(* CODESYS project Rasi_feeds_batching.project

Project tree, tasks and I/O mapping:
  PLC_AC500_V3 : PM5032-T-ETH, ABB AG, order no. 1SAP123400R0x72, version 3.7.0.0
    application Application
      task Task (cyclic, interval t#10ms, priority 14, watchdog t#20ms x 1) calls batching14
      CheckConfigurationObject
      old_version/
        program batching1 [ST]
        program batching2 [ST]
        program batching3 [ST]
        program batching4 [ST]
        program batching5 [ST]
        function block Auto_Batching [ST]
        function block Manual_Batching [ST]
        program batching6 [ST]
        function block Auto_Batching_V7 [ST]
        function block Manual_Batching_V7 [ST]
        program batching7 [ST]
        function block Auto_Batching_V8 [ST]
        function block Manual_Batching_V8 [ST]
        program batching8 [ST]
        function block Auto_Batching_V9 [ST]
        function block Manual_Batching_V9 [ST]
        program batching9 [ST]
        function block Auto_Batching_V10 [ST]
        function block Manual_Batching_V10 [ST]
        program batching10 [ST]
        program batching11 [ST]
        function block Auto_Batching_V11 [ST]
        function block Semi_Auto_Batching_V11 [ST]
        function block Auto_Batching_V12 [ST]
        function block Semi_Auto_Batching_V12 [ST]
        program batching12 [ST]
      Diagnosis/
        text list Diag_IO_Bus
        text list Diag_V3_PLC
      global variables GVL
      function block Auto_Batching_V13 [ST]
      function block Semi_Auto_Batching_V13 [ST]
      program batching13 [ST]
      function block Auto_Batching_V14 [ST]
      function block Semi_Auto_Batching_V14 [ST]
      program batching14 [FBD]
    OnBoard_IO : 12DI/8DO-T/2DC, ABB AG, version 3.7.0.0
        unmapped channels: Fast inputs DI0-DI3, Fast inputs DI4-DI7, Standard inputs DI8-DI11, Digital inputs - Transistor, Fast outputs DO0-DO3, Fast outputs DO4-DO7, Digital outputs - Transistor
    IO_Bus : I/O-Bus, ABB AG, version 3.7.0.0
    Interfaces : Interfaces, ABB AG, version 3.7.0.0
      OptionSlot_1
      OptionSlot_2
      Ethernet : Ethernet, ABB AG, version 3.7.0.0
        ETH1 : IP Settings, ABB AG, version 3.7.0.0
          NetConfig : NetConfig, ABB AG, version 3.7.0.0
          Modbus_TCP_IP_Server : Modbus TCP/IP Server, ABB AG, version 3.7.0.0
        Protocols : Client Protocols, ABB AG, version 3.7.0.0
    OnBoard_RTC : OnBoard RTC, ABB AG, version 3.7.0.0
  text list GlobalTextList
*)

// PLC_AC500_V3/Application/GVL
{attribute 'qualified_only'}
VAR_GLOBAL
    Recipe_Weights AT %MD100 : ARRAY[1..20] OF REAL;
	Auto_Bin_Material_Mapping AT %MW50: ARRAY[1..6] OF INT;
	Semi_Auto_Bin_Material_Mapping AT %MW60: ARRAY[1..10] OF INT;
	Auto_Bin_Cutoff_Weights AT %MD120: ARRAY[1..6] OF REAL;
	Semi_Auto_Bin_Cutoff_Weights AT %MD130: ARRAY[1..10] OF REAL;
	Auto_Bin_Tolerance AT %MD150: ARRAY[1..6] OF REAL;
	Semi_Auto_Bin_Tolerance AT %MD160: ARRAY[1..10] OF REAL;
	Start_Button AT %MX2.0: BOOL;
	E_Stop_Active AT %MX2.1: BOOL;
	Reset AT %MX2.3: BOOL;
	Cycle_Hold_Active AT %MX2.4: BOOL;
	Auto_Active_Mat AT %MW70: INT;
	Auto_Active_Bin AT %MW71: INT;
	Semi_Auto_Active_Mat AT %MW72: INT;
	Semi_Auto_Active_Bin AT %MW73: INT;
	Target_Batch_Cycles AT %MW74: INT;
	Current_Batch_Cycle AT %MW75: INT;
	Error_Code AT %MW76: INT;
	Run AT %MX2.5 : BOOL;
	load_cell_auto AT %MD174 : REAL;
	load_cell_semi_auto AT %MD175 : REAL;
	Auto_Initial_Tolerance AT %MD176 : REAL;
	Semi_Auto_Initial_Tolerance AT %MD178 : REAL;
	Auto_Total_Target_Weight AT %MD180 : REAL;
	Semi_Auto_Total_Target_Weight AT %MD184 : REAL;
	Auto_Material_Count AT %MW77 : INT;
	Semi_Auto_Material_Count AT %MW78 : INT;
	Auto_Current_Step AT %MW80 : INT;
	Semi_Auto_Current_Step AT %MW81 : INT;
	Auto_Active_Target_Weight AT %MD220 : REAL;
	Semi_Auto_Active_Target_Weight AT %MD224 : REAL;
	Auto_Active_Live_Weight AT %MD228 : REAL;
	Semi_Auto_Active_Live_Weight AT %MD232 : REAL;
	Auto_Excess_Allowed AT %MX2.6 : BOOL;
	Semi_Auto_Excess_Allowed AT %MX2.9 : BOOL;
	Auto_Excess_Alarm AT %MX2.7 : BOOL;
	Semi_Auto_Excess_Alarm AT %MX2.8 : BOOL;
	Auto_Inter_Bin_Delay AT %MD190 : TIME;
	Semi_Auto_Inter_Bin_Delay AT %MD194 : TIME;
	Auto_Sequence_Complete AT %MX3.0 : BOOL;
	Semi_Auto_Sequence_Complete AT %MX3.1 : BOOL;
	Auto_Status_Message : STRING(80);
	Semi_Auto_Status_Message : STRING(80);
	
	(* 8 Process Output and Weight Arrays *)
	Auto_Bin : ARRAY[1..6] OF BOOL;
	auto_bin_cutoff : ARRAY[1..6] OF BOOL;
	auto_bin_motor : ARRAY[1..6] OF BOOL;
	Semi_Auto_Bin : ARRAY[1..10] OF BOOL;
	semi_auto_bin_cutoff : ARRAY[1..10] OF BOOL;
	semi_auto_bin_motor : ARRAY[1..10] OF BOOL;
	Auto_Weights : ARRAY[1..6] OF REAL;
	Semi_Auto_Weights : ARRAY[1..10] OF REAL;
END_VAR

// PLC_AC500_V3/Application/batching14
PROGRAM batching14
VAR
	Auto_Ctrl: Auto_Batching_V14;
	Semi_Auto_Ctrl: Semi_Auto_Batching_V14;
	Auto_Complete: BOOL;
	Semi_Auto_Complete: BOOL;
	Auto_Err: INT;
	Semi_Auto_Err: INT;
END_VAR

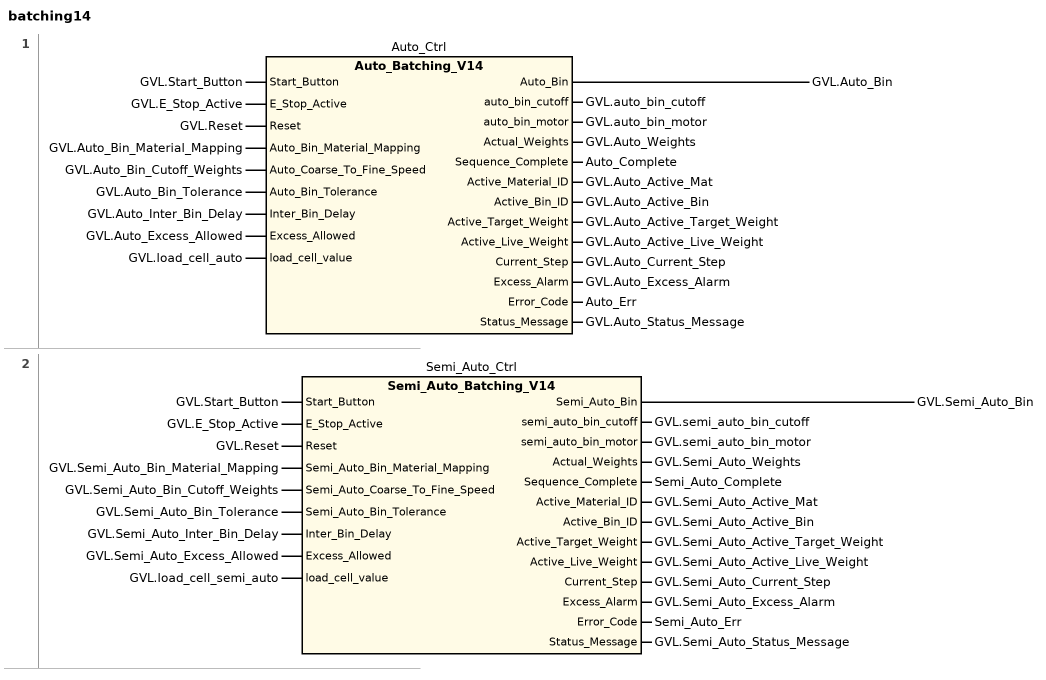
// NETWORK 1
Auto_Ctrl(
    Start_Button := GVL.Start_Button,
    E_Stop_Active := GVL.E_Stop_Active,
    Reset := GVL.Reset,
    Auto_Bin_Material_Mapping := GVL.Auto_Bin_Material_Mapping,
    Auto_Coarse_To_Fine_Speed := GVL.Auto_Bin_Cutoff_Weights,
    Auto_Bin_Tolerance := GVL.Auto_Bin_Tolerance,
    Inter_Bin_Delay := GVL.Auto_Inter_Bin_Delay,
    Excess_Allowed := GVL.Auto_Excess_Allowed,
    load_cell_value := GVL.load_cell_auto,
    auto_bin_cutoff => GVL.auto_bin_cutoff,
    auto_bin_motor => GVL.auto_bin_motor,
    Actual_Weights => GVL.Auto_Weights,
    Sequence_Complete => Auto_Complete,
    Active_Material_ID => GVL.Auto_Active_Mat,
    Active_Bin_ID => GVL.Auto_Active_Bin,
    Active_Target_Weight => GVL.Auto_Active_Target_Weight,
    Active_Live_Weight => GVL.Auto_Active_Live_Weight,
    Current_Step => GVL.Auto_Current_Step,
    Excess_Alarm => GVL.Auto_Excess_Alarm,
    Error_Code => Auto_Err,
    Status_Message => GVL.Auto_Status_Message); // Auto_Batching_V14
GVL.Auto_Bin := Auto_Ctrl.Auto_Bin;

// NETWORK 2
Semi_Auto_Ctrl(
    Start_Button := GVL.Start_Button,
    E_Stop_Active := GVL.E_Stop_Active,
    Reset := GVL.Reset,
    Semi_Auto_Bin_Material_Mapping := GVL.Semi_Auto_Bin_Material_Mapping,
    Semi_Auto_Coarse_To_Fine_Speed := GVL.Semi_Auto_Bin_Cutoff_Weights,
    Semi_Auto_Bin_Tolerance := GVL.Semi_Auto_Bin_Tolerance,
    Inter_Bin_Delay := GVL.Semi_Auto_Inter_Bin_Delay,
    Excess_Allowed := GVL.Semi_Auto_Excess_Allowed,
    load_cell_value := GVL.load_cell_semi_auto,
    semi_auto_bin_cutoff => GVL.semi_auto_bin_cutoff,
    semi_auto_bin_motor => GVL.semi_auto_bin_motor,
    Actual_Weights => GVL.Semi_Auto_Weights,
    Sequence_Complete => Semi_Auto_Complete,
    Active_Material_ID => GVL.Semi_Auto_Active_Mat,
    Active_Bin_ID => GVL.Semi_Auto_Active_Bin,
    Active_Target_Weight => GVL.Semi_Auto_Active_Target_Weight,
    Active_Live_Weight => GVL.Semi_Auto_Active_Live_Weight,
    Current_Step => GVL.Semi_Auto_Current_Step,
    Excess_Alarm => GVL.Semi_Auto_Excess_Alarm,
    Error_Code => Semi_Auto_Err,
    Status_Message => GVL.Semi_Auto_Status_Message); // Semi_Auto_Batching_V14
GVL.Semi_Auto_Bin := Semi_Auto_Ctrl.Semi_Auto_Bin;

END_PROGRAM

// PLC_AC500_V3/Application/Auto_Batching_V14
FUNCTION_BLOCK Auto_Batching_V14
VAR_INPUT
    Start_Button : BOOL;
    E_Stop_Active : BOOL;
    Reset : BOOL;
    Auto_Bin_Material_Mapping : ARRAY[1..6] OF INT;
    Auto_Coarse_To_Fine_Speed : ARRAY[1..6] OF REAL;
    Auto_Bin_Tolerance : ARRAY[1..6] OF REAL;
    Inter_Bin_Delay : TIME;
    Excess_Allowed : BOOL;
END_VAR
VAR_IN_OUT
    load_cell_value : REAL;
END_VAR
VAR_OUTPUT
    Auto_Bin : ARRAY[1..6] OF BOOL;
    auto_bin_cutoff : ARRAY[1..6] OF BOOL;
    auto_bin_motor : ARRAY[1..6] OF BOOL;
    Actual_Weights : ARRAY[1..6] OF REAL;
    Sequence_Complete : BOOL;
    Active_Material_ID : INT;
    Active_Bin_ID : INT;
    Active_Target_Weight : REAL;
    Active_Live_Weight : REAL;
    Current_Step : INT;
    Excess_Alarm : BOOL;
    Error_Code : INT;
    Status_Message : STRING(80);
END_VAR
VAR
    Step : INT;
    bin_last_weight : REAL;
    actual_bin : REAL;
    target_weight : REAL;
    cutoff_trigger_weight : REAL;
    min_tol_weight : REAL;
    max_tol_weight : REAL;
    Paused_By_EStop : BOOL;
    Effective_Delay : TIME;
    Mat_Idx : INT;
    i : INT;
    j : INT;
    Transition_Timer : TON;
    Completion_Timer : TON;
    Simulation_Mode : BOOL;
    Sim_Rate : REAL;
    Sim_Timer : TON;
    Start_Sim_Weight : REAL;
    Discharge_Active : BOOL;
    
    (* Master Cycle Manager & Supervisory states *)
    Cycle_Manager_State : INT;
    Internal_FB_Start : BOOL;
    Duplicate_Found : BOOL;
    Invalid_Material_Range : BOOL;
    Weight_Limit_Error : BOOL;
END_VAR

(* Auto Batching FB V14 with Full Diagnostics, Step Tracking, and Precise Status Reporting *)

Effective_Delay := Inter_Bin_Delay;
IF Effective_Delay = T#0S THEN
    Effective_Delay := T#2S;
END_IF;

(* Update Output Step *)
Current_Step := Step;

(* 1. RECIPE TOTALS & SUPERVISORY CONFIGURATION CHECKS *)
Duplicate_Found := FALSE;
Invalid_Material_Range := FALSE;
Weight_Limit_Error := FALSE;

GVL.Auto_Total_Target_Weight := 0.0;
GVL.Auto_Material_Count := 0;
FOR i := 1 TO 6 DO
    IF Auto_Bin_Material_Mapping[i] < 0 OR Auto_Bin_Material_Mapping[i] > 20 THEN
        Invalid_Material_Range := TRUE;
    END_IF;
    IF Auto_Bin_Material_Mapping[i] <> 0 AND Auto_Bin_Material_Mapping[i] <= 20 THEN
        FOR j := 1 TO 10 DO
            IF Auto_Bin_Material_Mapping[i] = GVL.Semi_Auto_Bin_Material_Mapping[j] THEN
                Duplicate_Found := TRUE;
            END_IF;
        END_FOR;
    END_IF;
    IF Auto_Bin_Material_Mapping[i] > 0 AND Auto_Bin_Material_Mapping[i] <= 20 THEN
        IF GVL.Recipe_Weights[Auto_Bin_Material_Mapping[i]] > 0.0 THEN
            GVL.Auto_Total_Target_Weight := GVL.Auto_Total_Target_Weight + GVL.Recipe_Weights[Auto_Bin_Material_Mapping[i]];
            GVL.Auto_Material_Count := GVL.Auto_Material_Count + 1;
            IF GVL.Recipe_Weights[Auto_Bin_Material_Mapping[i]] < (Auto_Coarse_To_Fine_Speed[i] + Auto_Bin_Tolerance[i]) THEN
                Weight_Limit_Error := TRUE;
            END_IF;
        END_IF;
    END_IF;
END_FOR;

IF Duplicate_Found THEN
    GVL.Error_Code := 1;
    Error_Code := 1;
    Status_Message := 'Error 1: Duplicate Material ID mapped in Auto and Semi-Auto!';
ELSIF Invalid_Material_Range THEN
    GVL.Error_Code := 2;
    Error_Code := 2;
    Status_Message := 'Error 2: Material Index configuration out of range (1..20)!';
ELSIF Weight_Limit_Error THEN
    GVL.Error_Code := 3;
    Error_Code := 3;
    Status_Message := 'Error 3: Recipe weight is less than Coarse_To_Fine_Speed + Tolerance!';
ELSE
    IF GVL.Error_Code <= 3 THEN
        GVL.Error_Code := 0;
        Error_Code := 0;
    END_IF;
END_IF;

(* 2. HARD RESET INTERLOCK *)
IF Reset OR GVL.Reset THEN
    FOR i := 1 TO 6 DO
        Auto_Bin[i] := FALSE;
        auto_bin_cutoff[i] := FALSE;
        auto_bin_motor[i] := FALSE;
        Actual_Weights[i] := 0.0;
        GVL.Auto_Bin[i] := FALSE;
        GVL.auto_bin_cutoff[i] := FALSE;
        GVL.auto_bin_motor[i] := FALSE;
        GVL.Auto_Weights[i] := 0.0;
    END_FOR;
    
    (* Reset Recipe & Active Target Setpoints *)
    FOR i := 1 TO 20 DO
        GVL.Recipe_Weights[i] := 0.0;
    END_FOR;
    GVL.Auto_Total_Target_Weight := 0.0;
    GVL.Semi_Auto_Total_Target_Weight := 0.0;
    GVL.Auto_Material_Count := 0;
    GVL.Semi_Auto_Material_Count := 0;
    
    Sequence_Complete := FALSE;
    GVL.Auto_Sequence_Complete := FALSE;
    GVL.Semi_Auto_Sequence_Complete := FALSE;
    Active_Material_ID := 0;
    Active_Bin_ID := 0;
    Active_Target_Weight := 0.0;
    Active_Live_Weight := 0.0;
    GVL.Auto_Active_Target_Weight := 0.0;
    GVL.Auto_Active_Live_Weight := 0.0;
    Excess_Alarm := FALSE;
    Error_Code := 0;
    GVL.Error_Code := 0;
    GVL.Current_Batch_Cycle := 0;
    GVL.Target_Batch_Cycles := 0;
    GVL.Start_Button := FALSE;
    GVL.Run := FALSE;
    GVL.Cycle_Hold_Active := FALSE;
    GVL.Auto_Active_Mat := 0;
    GVL.Auto_Active_Bin := 0;
    GVL.Auto_Excess_Alarm := FALSE;
    Step := 0;
    Current_Step := 0;
    Cycle_Manager_State := 0;
    Internal_FB_Start := FALSE;
    bin_last_weight := 0.0;
    Start_Sim_Weight := 0.0;
    Transition_Timer(IN := FALSE);
    Completion_Timer(IN := FALSE);
    Sim_Timer(IN := FALSE);
    Status_Message := 'Auto [Reset]: System Reset Complete - System Idle';
    RETURN;
END_IF;

(* 3. E-STOP PAUSE / HOLD LOGIC (NC Contact: FALSE = Pressed/Tripped, TRUE = Healthy) *)
IF NOT E_Stop_Active OR NOT GVL.E_Stop_Active THEN
    Paused_By_EStop := TRUE;
END_IF;

IF Paused_By_EStop THEN
    FOR i := 1 TO 6 DO
        Auto_Bin[i] := FALSE;
        auto_bin_cutoff[i] := FALSE;
        auto_bin_motor[i] := FALSE;
    END_FOR;
    IF NOT E_Stop_Active OR NOT GVL.E_Stop_Active THEN
        Status_Message := CONCAT('Auto [PAUSED]: E-Stop Active at Step ', INT_TO_STRING(Step));
    ELSE
        Status_Message := CONCAT('Auto [HOLD]: E-Stop Cleared. Press Start to Resume Step ', INT_TO_STRING(Step));
        IF Start_Button OR GVL.Start_Button THEN
            Paused_By_EStop := FALSE;
        END_IF;
    END_IF;
    Sim_Timer(IN := FALSE);
    Transition_Timer(IN := FALSE);
    Completion_Timer(IN := FALSE);
    RETURN;
END_IF;

(* 4. MASTER CYCLE MANAGER STATE MACHINE *)
CASE Cycle_Manager_State OF
    0: (* IDLE *)
        Internal_FB_Start := FALSE;
        GVL.Run := FALSE;
        GVL.Cycle_Hold_Active := FALSE;
        GVL.Auto_Sequence_Complete := FALSE;
        
        IF GVL.Error_Code = 0 THEN
            Status_Message := 'Auto [State 0 - Idle]: Ready - Waiting for Start Button';
        END_IF;
        
        IF Start_Button OR GVL.Start_Button THEN
            IF NOT E_Stop_Active OR NOT GVL.E_Stop_Active THEN
                GVL.Run := FALSE;
                Status_Message := 'Auto [State 0]: Cannot Start - Emergency Stop Contact Open!';
            ELSIF GVL.Target_Batch_Cycles <= 0 THEN
                GVL.Run := FALSE;
                Status_Message := 'Auto [State 0]: Cannot Start - Target Batch Cycles is 0!';
            ELSIF (GVL.load_cell_auto > GVL.Auto_Initial_Tolerance OR GVL.load_cell_auto < (-GVL.Auto_Initial_Tolerance)) OR 
                  (GVL.load_cell_semi_auto > GVL.Semi_Auto_Initial_Tolerance OR GVL.load_cell_semi_auto < (-GVL.Semi_Auto_Initial_Tolerance)) THEN
                GVL.Run := FALSE;
                GVL.Error_Code := 4;
                Error_Code := 4;
                Status_Message := 'Auto [State 0]: Error 4 - Scale weight exceeds Initial Tolerance!';
            ELSE
                GVL.Error_Code := 0;
                Error_Code := 0;
                GVL.Current_Batch_Cycle := 1;
                GVL.Run := TRUE;
                Internal_FB_Start := TRUE;
                Cycle_Manager_State := 1;
            END_IF;
        END_IF;
        
    1: (* RUNNING CYCLE *)
        Internal_FB_Start := TRUE;
        GVL.Run := TRUE;
        
        (* Both Auto and Semi-Auto must complete to finish the cycle *)
        IF Sequence_Complete AND GVL.Semi_Auto_Sequence_Complete THEN
            IF GVL.Current_Batch_Cycle < GVL.Target_Batch_Cycles AND GVL.Error_Code = 0 THEN
                GVL.Cycle_Hold_Active := TRUE;
                Internal_FB_Start := FALSE;
                Cycle_Manager_State := 5;
            ELSE
                Cycle_Manager_State := 4;
            END_IF;
        END_IF;
        
    5: (* PAUSED BETWEEN CYCLES IN HOLD *)
        Internal_FB_Start := FALSE;
        GVL.Run := TRUE;
        Status_Message := CONCAT('Auto [State 5 - Hold]: Cycle ', CONCAT(INT_TO_STRING(GVL.Current_Batch_Cycle), ' Complete. Empty scale to 0 and release Cycle Hold.'));
        
        IF NOT GVL.Cycle_Hold_Active THEN
            IF (GVL.load_cell_auto > GVL.Auto_Initial_Tolerance OR GVL.load_cell_auto < (-GVL.Auto_Initial_Tolerance)) OR 
               (GVL.load_cell_semi_auto > GVL.Semi_Auto_Initial_Tolerance OR GVL.load_cell_semi_auto < (-GVL.Semi_Auto_Initial_Tolerance)) THEN
                GVL.Run := FALSE;
                GVL.Error_Code := 4;
                Error_Code := 4;
                Status_Message := 'Auto [State 5]: Error 4 - Scale not zeroed! Tare scale before continuing.';
                GVL.Cycle_Hold_Active := TRUE;
            ELSE
                GVL.Error_Code := 0;
                Error_Code := 0;
                GVL.Current_Batch_Cycle := GVL.Current_Batch_Cycle + 1;
                Sequence_Complete := FALSE;
                GVL.Auto_Sequence_Complete := FALSE;
                GVL.Semi_Auto_Sequence_Complete := FALSE;
                Step := 0;
                Internal_FB_Start := TRUE;
                Cycle_Manager_State := 1;
            END_IF;
        END_IF;
        
    4: (* ALL CYCLES COMPLETE *)
        Internal_FB_Start := FALSE;
        GVL.Run := FALSE;
        GVL.Start_Button := FALSE;
        GVL.Auto_Sequence_Complete := FALSE;
        GVL.Semi_Auto_Sequence_Complete := FALSE;
        Status_Message := CONCAT('Auto [State 4 - Finished]: All ', CONCAT(INT_TO_STRING(GVL.Target_Batch_Cycles), ' Batch Cycles Completed Successfully'));
        Cycle_Manager_State := 0;
END_CASE;

(* 5. AUTO SILOS 1..6 POURING SEQUENCE WITH DETAILED STATUS *)
IF Step = 0 AND Internal_FB_Start THEN
    Step := 1;
    bin_last_weight := load_cell_value;
    Sequence_Complete := FALSE;
    GVL.Auto_Sequence_Complete := FALSE;
    Excess_Alarm := FALSE;
    Error_Code := 0;
    FOR i := 1 TO 6 DO
        Actual_Weights[i] := 0.0;
        Auto_Bin[i] := FALSE;
        auto_bin_cutoff[i] := FALSE;
        auto_bin_motor[i] := FALSE;
    END_FOR;
END_IF;

CASE Step OF
    0:
        Active_Material_ID := 0;
        Active_Bin_ID := 0;
        Excess_Alarm := FALSE;
        Sequence_Complete := FALSE;
        FOR i := 1 TO 6 DO
            Auto_Bin[i] := FALSE;
            auto_bin_cutoff[i] := FALSE;
            auto_bin_motor[i] := FALSE;
        END_FOR;
        Active_Target_Weight := GVL.Auto_Active_Target_Weight;
        Active_Live_Weight := 0.0;
        
    1..6:
        Mat_Idx := Auto_Bin_Material_Mapping[Step];
        
        IF (Mat_Idx = 0 OR (Mat_Idx <= 20 AND GVL.Recipe_Weights[Mat_Idx] = 0.0)) AND GVL.Auto_Active_Target_Weight = 0.0 THEN
            Status_Message := CONCAT('Auto [Step ', CONCAT(INT_TO_STRING(Step), ']: Silo Skipped (Target = 0)'));
            IF Step = 6 THEN
                Step := 7;
            ELSE
                Step := Step + 1;
            END_IF;
        ELSE
            IF Mat_Idx > 0 AND Mat_Idx <= 20 AND GVL.Recipe_Weights[Mat_Idx] > 0.0 THEN
                target_weight := GVL.Recipe_Weights[Mat_Idx];
            ELSE
                target_weight := GVL.Auto_Active_Target_Weight;
            END_IF;
            
            Active_Target_Weight := target_weight;
            GVL.Auto_Active_Target_Weight := target_weight;
            
            cutoff_trigger_weight := target_weight - Auto_Coarse_To_Fine_Speed[Step];
            min_tol_weight := target_weight - Auto_Bin_Tolerance[Step];
            max_tol_weight := target_weight + Auto_Bin_Tolerance[Step];
            
            actual_bin := load_cell_value - bin_last_weight;
            Actual_Weights[Step] := actual_bin;
            Active_Live_Weight := actual_bin;
            GVL.Auto_Active_Live_Weight := actual_bin;
            Active_Material_ID := Mat_Idx;
            Active_Bin_ID := Step;
            
            IF load_cell_value > 500.0 THEN
                Error_Code := 21;
                GVL.Error_Code := 21;
                Status_Message := CONCAT('Auto [Step ', CONCAT(INT_TO_STRING(Step), ']: STUCK - Error 21: Scale Overloaded (> 500 kg)!'));
                Sequence_Complete := TRUE;
                GVL.Auto_Sequence_Complete := TRUE;
                Paused_By_EStop := TRUE;
            END_IF;
            
            IF actual_bin < cutoff_trigger_weight THEN
                Auto_Bin[Step] := TRUE;
                auto_bin_cutoff[Step] := FALSE;
                auto_bin_motor[Step] := TRUE;
                Excess_Alarm := FALSE;
                Status_Message := CONCAT('Auto [Step ', CONCAT(INT_TO_STRING(Step), ']: Coarse Feeding'));
            ELSIF actual_bin < min_tol_weight THEN
                Auto_Bin[Step] := FALSE;
                auto_bin_cutoff[Step] := TRUE;
                auto_bin_motor[Step] := TRUE;
                Excess_Alarm := FALSE;
                Status_Message := CONCAT('Auto [Step ', CONCAT(INT_TO_STRING(Step), ']: Fine Feeding'));
            ELSIF actual_bin > max_tol_weight THEN
                Auto_Bin[Step] := FALSE;
                auto_bin_cutoff[Step] := FALSE;
                auto_bin_motor[Step] := FALSE;
                IF Excess_Allowed THEN
                    Excess_Alarm := FALSE;
                    Status_Message := CONCAT('Auto [Step ', CONCAT(INT_TO_STRING(Step), ']: Excess Allowed - Advancing'));
                    bin_last_weight := load_cell_value;
                    IF Step = 6 THEN
                        Step := 7;
                    ELSE
                        Step := Step + 1;
                    END_IF;
                ELSE
                    Excess_Alarm := TRUE;
                    Status_Message := CONCAT('Auto [Step ', CONCAT(INT_TO_STRING(Step), ']: STUCK - Excess Weight! Reduce weight or enable Excess Allowed.'));
                END_IF;
            ELSE
                Auto_Bin[Step] := FALSE;
                auto_bin_cutoff[Step] := FALSE;
                auto_bin_motor[Step] := FALSE;
                Excess_Alarm := FALSE;
                bin_last_weight := load_cell_value;
                Status_Message := CONCAT('Auto [Step ', CONCAT(INT_TO_STRING(Step), ']: Target Reached - Advancing'));
                IF Step = 6 THEN
                    Step := 7;
                ELSE
                    Step := Step + 1;
                END_IF;
            END_IF;
        END_IF;

    7:
        Active_Material_ID := 0;
        Active_Bin_ID := 0;
        Excess_Alarm := FALSE;
        Status_Message := 'Auto [Step 7]: Settling Delay in progress...';
        Completion_Timer(IN := TRUE, PT := Effective_Delay);
        IF Completion_Timer.Q THEN
            Completion_Timer(IN := FALSE);
            Step := 8;
        END_IF;
        
    8:
        Active_Material_ID := 0;
        Active_Bin_ID := 0;
        Excess_Alarm := FALSE;
        Sequence_Complete := TRUE;
        GVL.Auto_Sequence_Complete := TRUE;
        IF NOT GVL.Semi_Auto_Sequence_Complete THEN
            Status_Message := 'Auto [Step 8]: Auto Finished. Waiting for Semi-Auto to complete...';
        ELSE
            Status_Message := 'Auto [Step 8]: Cycle Sequences Complete';
        END_IF;
        
        IF NOT Internal_FB_Start THEN
            Step := 0;
            Sequence_Complete := FALSE;
            GVL.Auto_Sequence_Complete := FALSE;
            FOR i := 1 TO 6 DO
                Actual_Weights[i] := 0.0;
            END_FOR;
        END_IF;
END_CASE;

END_FUNCTION_BLOCK

// PLC_AC500_V3/Application/Semi_Auto_Batching_V14
FUNCTION_BLOCK Semi_Auto_Batching_V14
VAR_INPUT
    Start_Button : BOOL;
    E_Stop_Active : BOOL;
    Reset : BOOL;
    Semi_Auto_Bin_Material_Mapping : ARRAY[1..10] OF INT;
    Semi_Auto_Coarse_To_Fine_Speed : ARRAY[1..10] OF REAL;
    Semi_Auto_Bin_Tolerance : ARRAY[1..10] OF REAL;
    Inter_Bin_Delay : TIME;
    Excess_Allowed : BOOL;
END_VAR
VAR_IN_OUT
    load_cell_value : REAL;
END_VAR
VAR_OUTPUT
    Semi_Auto_Bin : ARRAY[1..10] OF BOOL;
    semi_auto_bin_cutoff : ARRAY[1..10] OF BOOL;
    semi_auto_bin_motor : ARRAY[1..10] OF BOOL;
    Actual_Weights : ARRAY[1..10] OF REAL;
    Sequence_Complete : BOOL;
    Active_Material_ID : INT;
    Active_Bin_ID : INT;
    Active_Target_Weight : REAL;
    Active_Live_Weight : REAL;
    Current_Step : INT;
    Excess_Alarm : BOOL;
    Error_Code : INT;
    Status_Message : STRING(80);
END_VAR
VAR
    Step : INT;
    bin_last_weight : REAL;
    actual_bin : REAL;
    target_weight : REAL;
    cutoff_trigger_weight : REAL;
    min_tol_weight : REAL;
    max_tol_weight : REAL;
    Paused_By_EStop : BOOL;
    Effective_Delay : TIME;
    Mat_Idx : INT;
    i : INT;
    Transition_Timer : TON;
    Completion_Timer : TON;
    Simulation_Mode : BOOL;
    Sim_Rate : REAL;
    Sim_Timer : TON;
    Start_Sim_Weight : REAL;
    Discharge_Active : BOOL;
END_VAR

(* Semi-Auto Batching FB V14 with Full Diagnostics, Step Tracking, and Precise Status Reporting *)

Effective_Delay := Inter_Bin_Delay;
IF Effective_Delay = T#0S THEN
    Effective_Delay := T#2S;
END_IF;

(* Update Output Step *)
Current_Step := Step;

(* 1. SEMI-AUTO RECIPE TOTALS & ACTIVE SILO COUNT *)
GVL.Semi_Auto_Total_Target_Weight := 0.0;
GVL.Semi_Auto_Material_Count := 0;
FOR i := 1 TO 10 DO
    IF Semi_Auto_Bin_Material_Mapping[i] > 0 AND Semi_Auto_Bin_Material_Mapping[i] <= 20 THEN
        IF GVL.Recipe_Weights[Semi_Auto_Bin_Material_Mapping[i]] > 0.0 THEN
            GVL.Semi_Auto_Total_Target_Weight := GVL.Semi_Auto_Total_Target_Weight + GVL.Recipe_Weights[Semi_Auto_Bin_Material_Mapping[i]];
            GVL.Semi_Auto_Material_Count := GVL.Semi_Auto_Material_Count + 1;
        END_IF;
    END_IF;
END_FOR;

(* 2. HARD RESET INTERLOCK *)
IF Reset OR GVL.Reset THEN
    FOR i := 1 TO 10 DO
        Semi_Auto_Bin[i] := FALSE;
        semi_auto_bin_cutoff[i] := FALSE;
        semi_auto_bin_motor[i] := FALSE;
        Actual_Weights[i] := 0.0;
        GVL.Semi_Auto_Bin[i] := FALSE;
        GVL.semi_auto_bin_cutoff[i] := FALSE;
        GVL.semi_auto_bin_motor[i] := FALSE;
        GVL.Semi_Auto_Weights[i] := 0.0;
    END_FOR;
    Sequence_Complete := FALSE;
    GVL.Semi_Auto_Sequence_Complete := FALSE;
    Active_Material_ID := 0;
    Active_Bin_ID := 0;
    Active_Target_Weight := 0.0;
    Active_Live_Weight := 0.0;
    GVL.Semi_Auto_Active_Target_Weight := 0.0;
    GVL.Semi_Auto_Active_Live_Weight := 0.0;
    GVL.Semi_Auto_Active_Mat := 0;
    GVL.Semi_Auto_Active_Bin := 0;
    GVL.Semi_Auto_Excess_Alarm := FALSE;
    Excess_Alarm := FALSE;
    Error_Code := 0;
    Paused_By_EStop := FALSE;
    Step := 0;
    Current_Step := 0;
    bin_last_weight := 0.0;
    Start_Sim_Weight := 0.0;
    Transition_Timer(IN := FALSE);
    Completion_Timer(IN := FALSE);
    Sim_Timer(IN := FALSE);
    Status_Message := 'Semi-Auto [Reset]: System Reset Complete - System Idle';
    
    (* Clean Auto-Clearing: Reset has been processed by both blocks *)
    GVL.Reset := FALSE;
    RETURN;
END_IF;

(* 3. E-STOP PAUSE / HOLD LOGIC (NC Contact: FALSE = Pressed/Tripped, TRUE = Healthy) *)
IF NOT E_Stop_Active OR NOT GVL.E_Stop_Active THEN
    Paused_By_EStop := TRUE;
END_IF;

IF Paused_By_EStop THEN
    FOR i := 1 TO 10 DO
        Semi_Auto_Bin[i] := FALSE;
        semi_auto_bin_cutoff[i] := FALSE;
        semi_auto_bin_motor[i] := FALSE;
    END_FOR;
    IF NOT E_Stop_Active OR NOT GVL.E_Stop_Active THEN
        Status_Message := CONCAT('Semi-Auto [PAUSED]: E-Stop Active at Step ', INT_TO_STRING(Step));
    ELSE
        Status_Message := CONCAT('Semi-Auto [HOLD]: E-Stop Cleared. Press Start to Resume Step ', INT_TO_STRING(Step));
        IF Start_Button OR GVL.Start_Button THEN
            Paused_By_EStop := FALSE;
        END_IF;
    END_IF;
    Sim_Timer(IN := FALSE);
    Transition_Timer(IN := FALSE);
    Completion_Timer(IN := FALSE);
    RETURN;
END_IF;

(* 4. CYCLE HOLD RESET *)
IF GVL.Cycle_Hold_Active THEN
    Step := 0;
    Sequence_Complete := FALSE;
    GVL.Semi_Auto_Sequence_Complete := FALSE;
    Status_Message := 'Semi-Auto [Cycle Hold]: Waiting for next cycle...';
END_IF;

(* 5. SEQUENCE START (WHEN SYSTEM IS IN RUN MODE) *)
IF Step = 0 AND (GVL.Run OR Start_Button) AND GVL.Cycle_Hold_Active = FALSE AND NOT GVL.Semi_Auto_Sequence_Complete THEN
    Step := 1;
    bin_last_weight := load_cell_value;
    Sequence_Complete := FALSE;
    GVL.Semi_Auto_Sequence_Complete := FALSE;
    Excess_Alarm := FALSE;
    Error_Code := 0;
    FOR i := 1 TO 10 DO
        Actual_Weights[i] := 0.0;
        Semi_Auto_Bin[i] := FALSE;
        semi_auto_bin_cutoff[i] := FALSE;
        semi_auto_bin_motor[i] := FALSE;
    END_FOR;
END_IF;

CASE Step OF
    0:
        Active_Material_ID := 0;
        Active_Bin_ID := 0;
        Excess_Alarm := FALSE;
        Sequence_Complete := FALSE;
        FOR i := 1 TO 10 DO
            Semi_Auto_Bin[i] := FALSE;
            semi_auto_bin_cutoff[i] := FALSE;
            semi_auto_bin_motor[i] := FALSE;
        END_FOR;
        Active_Target_Weight := GVL.Semi_Auto_Active_Target_Weight;
        Active_Live_Weight := 0.0;
        IF Error_Code = 0 AND NOT GVL.Cycle_Hold_Active THEN 
            Status_Message := 'Semi-Auto [Step 0 - Idle]: Ready - Waiting for Run Signal'; 
        END_IF;
        
    1..10:
        Mat_Idx := Semi_Auto_Bin_Material_Mapping[Step];
        
        IF (Mat_Idx = 0 OR (Mat_Idx <= 20 AND GVL.Recipe_Weights[Mat_Idx] = 0.0)) AND GVL.Semi_Auto_Active_Target_Weight = 0.0 THEN
            Status_Message := CONCAT('Semi-Auto [Step ', CONCAT(INT_TO_STRING(Step), ']: Silo Skipped (Target = 0)'));
            IF Step = 10 THEN
                Step := 31;
            ELSE
                Step := Step + 1;
            END_IF;
        ELSE
            IF Mat_Idx > 0 AND Mat_Idx <= 20 AND GVL.Recipe_Weights[Mat_Idx] > 0.0 THEN
                target_weight := GVL.Recipe_Weights[Mat_Idx];
            ELSE
                target_weight := GVL.Semi_Auto_Active_Target_Weight;
            END_IF;
            
            Active_Target_Weight := target_weight;
            GVL.Semi_Auto_Active_Target_Weight := target_weight;
            
            cutoff_trigger_weight := target_weight - Semi_Auto_Coarse_To_Fine_Speed[Step];
            min_tol_weight := target_weight - Semi_Auto_Bin_Tolerance[Step];
            max_tol_weight := target_weight + Semi_Auto_Bin_Tolerance[Step];
            
            actual_bin := load_cell_value - bin_last_weight;
            Actual_Weights[Step] := actual_bin;
            Active_Live_Weight := actual_bin;
            GVL.Semi_Auto_Active_Live_Weight := actual_bin;
            Active_Material_ID := Mat_Idx;
            Active_Bin_ID := Step;
            
            IF load_cell_value > 500.0 THEN
                Error_Code := 21;
                GVL.Error_Code := 21;
                Status_Message := CONCAT('Semi-Auto [Step ', CONCAT(INT_TO_STRING(Step), ']: STUCK - Error 21: Scale Overloaded (> 500 kg)!'));
                Sequence_Complete := TRUE;
                GVL.Semi_Auto_Sequence_Complete := TRUE;
                Paused_By_EStop := TRUE;
            END_IF;
            
            IF actual_bin < cutoff_trigger_weight THEN
                Semi_Auto_Bin[Step] := TRUE;
                semi_auto_bin_cutoff[Step] := FALSE;
                semi_auto_bin_motor[Step] := TRUE;
                Excess_Alarm := FALSE;
                Status_Message := CONCAT('Semi-Auto [Step ', CONCAT(INT_TO_STRING(Step), ']: Coarse Feeding'));
            ELSIF actual_bin < min_tol_weight THEN
                Semi_Auto_Bin[Step] := FALSE;
                semi_auto_bin_cutoff[Step] := TRUE;
                semi_auto_bin_motor[Step] := TRUE;
                Excess_Alarm := FALSE;
                Status_Message := CONCAT('Semi-Auto [Step ', CONCAT(INT_TO_STRING(Step), ']: Fine Feeding'));
            ELSIF actual_bin > max_tol_weight THEN
                Semi_Auto_Bin[Step] := FALSE;
                semi_auto_bin_cutoff[Step] := FALSE;
                semi_auto_bin_motor[Step] := FALSE;
                IF Excess_Allowed THEN
                    Excess_Alarm := FALSE;
                    Status_Message := CONCAT('Semi-Auto [Step ', CONCAT(INT_TO_STRING(Step), ']: Excess Allowed - Advancing'));
                    bin_last_weight := load_cell_value;
                    IF Step = 10 THEN
                        Step := 31;
                    ELSE
                        Step := Step + 1;
                    END_IF;
                ELSE
                    Excess_Alarm := TRUE;
                    Status_Message := CONCAT('Semi-Auto [Step ', CONCAT(INT_TO_STRING(Step), ']: STUCK - Excess Weight! Reduce weight or enable Excess Allowed.'));
                END_IF;
            ELSE
                Semi_Auto_Bin[Step] := FALSE;
                semi_auto_bin_cutoff[Step] := FALSE;
                semi_auto_bin_motor[Step] := FALSE;
                Excess_Alarm := FALSE;
                bin_last_weight := load_cell_value;
                Status_Message := CONCAT('Semi-Auto [Step ', CONCAT(INT_TO_STRING(Step), ']: Target Reached - Advancing'));
                IF Step = 10 THEN
                    Step := 31;
                ELSE
                    Step := Step + 1;
                END_IF;
            END_IF;
        END_IF;

    31:
        Active_Material_ID := 0;
        Active_Bin_ID := 0;
        Excess_Alarm := FALSE;
        Status_Message := 'Semi-Auto [Step 31]: Settling Delay in progress...';
        Completion_Timer(IN := TRUE, PT := Effective_Delay);
        IF Completion_Timer.Q THEN
            Completion_Timer(IN := FALSE);
            Step := 32;
        END_IF;
        
    32:
        Active_Material_ID := 0;
        Active_Bin_ID := 0;
        Excess_Alarm := FALSE;
        Sequence_Complete := TRUE;
        GVL.Semi_Auto_Sequence_Complete := TRUE;
        IF NOT GVL.Auto_Sequence_Complete THEN
            Status_Message := 'Semi-Auto [Step 32]: Semi-Auto Finished. Waiting for Auto to complete...';
        ELSE
            Status_Message := 'Semi-Auto [Step 32]: Cycle Sequences Complete';
        END_IF;
        
        IF NOT GVL.Run THEN
            Step := 0;
            Sequence_Complete := FALSE;
            GVL.Semi_Auto_Sequence_Complete := FALSE;
            FOR i := 1 TO 10 DO
                Actual_Weights[i] := 0.0;
            END_FOR;
        END_IF;
END_CASE;

END_FUNCTION_BLOCK

// PLC_AC500_V3/Application/old_version/batching1
PROGRAM batching1
VAR
    Step : INT := 0;
    
    (* Mode Control *)
    Auto_Mode : BOOL := TRUE; // TRUE for Auto, FALSE for Manual
    
    (* Control Buttons *)
    Start_Button : BOOL;      // Start button for Auto sequence
    E_Stop_Active : BOOL;     // Emergency Stop active signal (normally open logic in software)
    
    (* Manual Buttons *)
    Manual_Bin1 : BOOL;       // Manual discharge trigger for Bin 1
    Manual_Bin2 : BOOL;       // Manual discharge trigger for Bin 2
    Manual_Bin3 : BOOL;       // Manual discharge trigger for Bin 3
    
    (* Discharge outputs *)
    Discharge_Bin1 : BOOL;
    Discharge_Bin2 : BOOL;
    Discharge_Bin3 : BOOL;
    
    (* Valve feedback (set to TRUE when open, FALSE when closed) *)
    Discharge_Bin1_Feedback : BOOL;
    Discharge_Bin2_Feedback : BOOL;
    Discharge_Bin3_Feedback : BOOL;
    
    (* Empty status / feedback *)
    Bin1_Empty : BOOL;
    Bin2_Empty : BOOL;
    Bin3_Empty : BOOL;
    
    (* Weight sensors (optional feedback) *)
    Bin1_Weight : REAL;
    Bin2_Weight : REAL;
    Bin3_Weight : REAL;
    
    Sequence_Complete : BOOL;
    
    (* DELAYS FOR VISUAL MONITORING *)
    Bin3_Timer : TON;         // Timer for Bin 3 discharge
    Bin2_Timer : TON;         // Timer for Bin 2 discharge
    Bin1_Timer : TON;         // Timer for Bin 1 discharge
    Transition_Timer : TON;   // Timer for transitions between stages
    
    Min_Discharge_Time : TIME := T#3S;  // Minimum time each bin stays open to allow visibility (e.g. 3 seconds)
    Step_Delay_Time : TIME := T#2S;     // Wait time between closing one bin and opening the next (e.g. 2 seconds)
END_VAR

(* Discharging Sequence with Auto/Manual Mode, E-Stop, Manual Controls, and Monitoring Delays *)

(* Emergency Stop Logic - High Priority *)
IF E_Stop_Active THEN
    Discharge_Bin1 := FALSE;
    Discharge_Bin2 := FALSE;
    Discharge_Bin3 := FALSE;
    Sequence_Complete := FALSE;
    Step := 0;
    
    (* Reset Timers *)
    Bin3_Timer(IN := FALSE);
    Bin2_Timer(IN := FALSE);
    Bin1_Timer(IN := FALSE);
    Transition_Timer(IN := FALSE);
    RETURN; // Halt execution of the rest of the POU
END_IF;

(* Mode Selection *)
IF Auto_Mode THEN
    (* ================= AUTOMATIC MODE ================= *)
    CASE Step OF
        0: (* Idle state *)
            Discharge_Bin1 := FALSE;
            Discharge_Bin2 := FALSE;
            Discharge_Bin3 := FALSE;
            Sequence_Complete := FALSE;
            
            Bin3_Timer(IN := FALSE);
            Bin2_Timer(IN := FALSE);
            Bin1_Timer(IN := FALSE);
            Transition_Timer(IN := FALSE);
            
            IF Start_Button THEN
                Step := 10;
            END_IF
            
        10: (* Discharge Bin 3 - ON *)
            Discharge_Bin3 := TRUE;
            Discharge_Bin2 := FALSE;
            Discharge_Bin1 := FALSE;
            
            (* Run timer to ensure discharge is visible *)
            Bin3_Timer(IN := TRUE, PT := Min_Discharge_Time);
            
            (* Transition when empty AND minimum time has elapsed *)
            IF (Bin3_Empty OR Bin3_Weight <= 0) AND Bin3_Timer.Q THEN
                Bin3_Timer(IN := FALSE); // Reset timer
                Step := 15;
            END_IF
            
        15: (* Discharge Bin 3 - OFF & Wait Transition Delay *)
            Discharge_Bin3 := FALSE;
            Transition_Timer(IN := TRUE, PT := Step_Delay_Time);
            
            IF Transition_Timer.Q AND (NOT Discharge_Bin3_Feedback OR NOT Discharge_Bin3) THEN
                Transition_Timer(IN := FALSE); // Reset timer
                Step := 20;
            END_IF
            
        20: (* Discharge Bin 2 - ON *)
            Discharge_Bin2 := TRUE;
            Discharge_Bin3 := FALSE;
            Discharge_Bin1 := FALSE;
            
            Bin2_Timer(IN := TRUE, PT := Min_Discharge_Time);
            
            IF (Bin2_Empty OR Bin2_Weight <= 0) AND Bin2_Timer.Q THEN
                Bin2_Timer(IN := FALSE);
                Step := 25;
            END_IF
            
        25: (* Discharge Bin 2 - OFF & Wait Transition Delay *)
            Discharge_Bin2 := FALSE;
            Transition_Timer(IN := TRUE, PT := Step_Delay_Time);
            
            IF Transition_Timer.Q AND (NOT Discharge_Bin2_Feedback OR NOT Discharge_Bin2) THEN
                Transition_Timer(IN := FALSE);
                Step := 30;
            END_IF
            
        30: (* Discharge Bin 1 - ON *)
            Discharge_Bin1 := TRUE;
            Discharge_Bin3 := FALSE;
            Discharge_Bin2 := FALSE;
            
            Bin1_Timer(IN := TRUE, PT := Min_Discharge_Time);
            
            IF (Bin1_Empty OR Bin1_Weight <= 0) AND Bin1_Timer.Q THEN
                Bin1_Timer(IN := FALSE);
                Step := 35;
            END_IF
            
        35: (* Discharge Bin 1 - OFF & Wait Transition Delay *)
            Discharge_Bin1 := FALSE;
            Transition_Timer(IN := TRUE, PT := Step_Delay_Time);
            
            IF Transition_Timer.Q AND (NOT Discharge_Bin1_Feedback OR NOT Discharge_Bin1) THEN
                Transition_Timer(IN := FALSE);
                Step := 40;
            END_IF
            
        40: (* Sequence Complete *)
            Sequence_Complete := TRUE;
            IF NOT Start_Button THEN
                Step := 0;
            END_IF
    END_CASE;

ELSE
    (* ================= MANUAL MODE ================= *)
    Step := 0;
    Sequence_Complete := FALSE;
    
    (* Reset all timers *)
    Bin3_Timer(IN := FALSE);
    Bin2_Timer(IN := FALSE);
    Bin1_Timer(IN := FALSE);
    Transition_Timer(IN := FALSE);
    
    (* Separate buttons for each bin with interlinking *)
    IF Manual_Bin3 THEN
        Discharge_Bin3 := TRUE;
        Discharge_Bin2 := FALSE;
        Discharge_Bin1 := FALSE;
    ELSIF Manual_Bin2 THEN
        Discharge_Bin3 := FALSE;
        Discharge_Bin2 := TRUE;
        Discharge_Bin1 := FALSE;
    ELSIF Manual_Bin1 THEN
        Discharge_Bin3 := FALSE;
        Discharge_Bin2 := FALSE;
        Discharge_Bin1 := TRUE;
    ELSE
        Discharge_Bin3 := FALSE;
        Discharge_Bin2 := FALSE;
        Discharge_Bin1 := FALSE;
    END_IF;
END_IF;

END_PROGRAM

// PLC_AC500_V3/Application/old_version/batching2
PROGRAM batching2
VAR
    Step : INT := 0;
    
    (* Mode Control *)
    Auto_Mode : BOOL := TRUE; // TRUE for Auto, FALSE for Manual
    Simulation_Mode : BOOL := TRUE; // Set to TRUE for software simulation, FALSE for physical hardware
    
    (* Control Buttons *)
    Start_Button : BOOL;      // Start button for Auto sequence
    E_Stop_Active : BOOL;     // Emergency Stop active signal
    
    (* Manual Buttons *)
    Manual_Bin1 : BOOL;       // Manual discharge trigger for Bin 1
    Manual_Bin2 : BOOL;       // Manual discharge trigger for Bin 2
    Manual_Bin3 : BOOL;       // Manual discharge trigger for Bin 3
    
    (* Discharge outputs *)
    Discharge_Bin1 : BOOL;
    Discharge_Bin2 : BOOL;
    Discharge_Bin3 : BOOL;
    
    (* Valve feedback *)
    Discharge_Bin1_Feedback : BOOL;
    Discharge_Bin2_Feedback : BOOL;
    Discharge_Bin3_Feedback : BOOL;
    
    (* Modbus Weight Inputs (Current Weight of the Bins) *)
    Current_Weight_Bin1 : REAL; // Current load cell reading for Bin 1 (Water)
    Current_Weight_Bin2 : REAL; // Current load cell reading for Bin 2 (Aggregate)
    Current_Weight_Bin3 : REAL; // Current load cell reading for Bin 3 (Cement)
    
    (* Starting Weights (Captured at start of process) *)
    Start_Weight_Bin1 : REAL;   // Weight snapshot of Bin 1 at start
    Start_Weight_Bin2 : REAL;   // Weight snapshot of Bin 2 at start
    Start_Weight_Bin3 : REAL;   // Weight snapshot of Bin 3 at start
    
    (* Target Discharge Threshold Amounts *)
    Target_Amount_Bin1 : REAL := 0.5;  // Amount of Water to discharge (e.g. 0.5 L)
    Target_Amount_Bin2 : REAL := 1.5;  // Amount of Aggregate to discharge (e.g. 1.5 kg)
    Target_Amount_Bin3 : REAL := 1.0;  // Amount of Cement to discharge (e.g. 1.0 kg)
    
    (* Calculated Cutoff Weights *)
    Cutoff_Weight_Bin1 : REAL;
    Cutoff_Weight_Bin2 : REAL;
    Cutoff_Weight_Bin3 : REAL;
    
    Sequence_Complete : BOOL;
    Transition_Timer : TON;
    Step_Delay_Time : TIME := T#2S;     // Delay between closing one valve and opening the next
    
    (* TIMERS FOR WEIGHT DECREMENT (EXACT 1.0 kg/s SIMULATION) *)
    Bin3_Timer : TON;         // Tracks elapsed open time of Bin 3
    Bin2_Timer : TON;         // Tracks elapsed open time of Bin 2
    Bin1_Timer : TON;         // Tracks elapsed open time of Bin 1
    
    (* SIMULATION DISCHARGE RATES (units per second) *)
    Sim_Rate_Bin1 : REAL := 1.0;        // Water loss rate: 1.0 L / second
    Sim_Rate_Bin2 : REAL := 1.0;        // Aggregate loss rate: 1.0 kg / second
    Sim_Rate_Bin3 : REAL := 1.0;        // Cement loss rate: 1.0 kg / second
    
    (* Modbus Master instances for each load cell (Commented out for compile-safety in simulation) *)
    (*
    Read_LC1 : COM_MODMAST;
    Read_LC2 : COM_MODMAST;
    Read_LC3 : COM_MODMAST;
    *)
    
    (* Modbus buffers (Commented out for compile-safety in simulation) *)
    (*
    LC1_Buffer : ARRAY[0..1] OF WORD;
    LC2_Buffer : ARRAY[0..1] OF WORD;
    LC3_Buffer : ARRAY[0..1] OF WORD;
    *)
END_VAR

(* Discharging Sequence with Auto/Manual Mode, E-Stop, Manual Controls, and Loss-in-Weight Threshold Cutoffs *)

(* 1. SIMULATION LOGIC (To run without physical Modbus hardware) *)
IF Simulation_Mode THEN
    (* Initialize weights to start values in Idle state *)
    IF Step = 0 AND NOT Start_Button AND NOT Sequence_Complete THEN
        Current_Weight_Bin3 := 70.0; // 70 kg Cement
        Current_Weight_Bin2 := 50.0; // 50 kg Aggregate
        Current_Weight_Bin1 := 80.0; // 80 L Water
    END_IF;
    
    (* Dynamically reduce weights based on elapsed time of active discharge (scan-time independent) *)
    IF Discharge_Bin3 THEN
        Bin3_Timer(IN := TRUE, PT := T#1000S);
        Current_Weight_Bin3 := Start_Weight_Bin3 - (TIME_TO_REAL(Bin3_Timer.ET) / 1000.0) * Sim_Rate_Bin3;
    ELSE
        Bin3_Timer(IN := FALSE);
    END_IF;
    
    IF Discharge_Bin2 THEN
        Bin2_Timer(IN := TRUE, PT := T#1000S);
        Current_Weight_Bin2 := Start_Weight_Bin2 - (TIME_TO_REAL(Bin2_Timer.ET) / 1000.0) * Sim_Rate_Bin2;
    ELSE
        Bin2_Timer(IN := FALSE);
    END_IF;
    
    IF Discharge_Bin1 THEN
        Bin1_Timer(IN := TRUE, PT := T#1000S);
        Current_Weight_Bin1 := Start_Weight_Bin1 - (TIME_TO_REAL(Bin1_Timer.ET) / 1000.0) * Sim_Rate_Bin1;
    ELSE
        Bin1_Timer(IN := FALSE);
    END_IF;
ELSE
    (* ================= PHYSICAL MODBUS RTU DATA ACQUISITION ================= *)
    (* Uncomment these blocks and their declarations when deploying to physical hardware *)
    (*
    Read_LC1(
        EN := TRUE,
        COM := 1,
        SLV := 1,
        FCT := 3,
        ADDR := 40001,
        SZ := 2,
        DATA := ADR(LC1_Buffer)
    );
    Current_Weight_Bin1 := WORD_TO_REAL(LC1_Buffer[0]);
    
    Read_LC2(
        EN := TRUE,
        COM := 1,
        SLV := 2,
        FCT := 3,
        ADDR := 40001,
        SZ := 2,
        DATA := ADR(LC2_Buffer)
    );
    Current_Weight_Bin2 := WORD_TO_REAL(LC2_Buffer[0]);
    
    Read_LC3(
        EN := TRUE,
        COM := 1,
        SLV := 3,
        FCT := 3,
        ADDR := 40001,
        SZ := 2,
        DATA := ADR(LC3_Buffer)
    );
    Current_Weight_Bin3 := WORD_TO_REAL(LC3_Buffer[0]);
    *)
END_IF;


(* 2. EMERGENCY STOP LOGIC *)
IF E_Stop_Active THEN
    Discharge_Bin1 := FALSE;
    Discharge_Bin2 := FALSE;
    Discharge_Bin3 := FALSE;
    Sequence_Complete := FALSE;
    Step := 0;
    Transition_Timer(IN := FALSE);
    RETURN;
END_IF;


(* 3. SEQUENCE CONTROL *)
IF Auto_Mode THEN
    (* ================= AUTOMATIC MODE ================= *)
    CASE Step OF
        0: (* Idle state *)
            Discharge_Bin1 := FALSE;
            Discharge_Bin2 := FALSE;
            Discharge_Bin3 := FALSE;
            Sequence_Complete := FALSE;
            Transition_Timer(IN := FALSE);
            
            IF Start_Button THEN
                (* Take snapshot of initial load cell weights *)
                Start_Weight_Bin1 := Current_Weight_Bin1;
                Start_Weight_Bin2 := Current_Weight_Bin2;
                Start_Weight_Bin3 := Current_Weight_Bin3;
                
                (* Calculate required cutoff weights based on discharge thresholds *)
                Cutoff_Weight_Bin3 := Start_Weight_Bin3 - Target_Amount_Bin3;
                Cutoff_Weight_Bin2 := Start_Weight_Bin2 - Target_Amount_Bin2;
                Cutoff_Weight_Bin1 := Start_Weight_Bin1 - Target_Amount_Bin1;
                
                Step := 10;
            END_IF
            
        10: (* Discharge Bin 3 - ON *)
            Discharge_Bin3 := TRUE;
            Discharge_Bin2 := FALSE;
            Discharge_Bin1 := FALSE;
            
            (* Check if current weight has dropped below target cutoff *)
            IF Current_Weight_Bin3 <= Cutoff_Weight_Bin3 THEN
                Step := 15;
            END_IF
            
        15: (* Discharge Bin 3 - OFF & Wait Transition Delay *)
            Discharge_Bin3 := FALSE;
            Transition_Timer(IN := TRUE, PT := Step_Delay_Time);
            
            IF Transition_Timer.Q AND (NOT Discharge_Bin3_Feedback OR NOT Discharge_Bin3) THEN
                Transition_Timer(IN := FALSE);
                Step := 20;
            END_IF
            
        20: (* Discharge Bin 2 - ON *)
            Discharge_Bin2 := TRUE;
            Discharge_Bin3 := FALSE;
            Discharge_Bin1 := FALSE;
            
            (* Check if current weight has dropped below target cutoff *)
            IF Current_Weight_Bin2 <= Cutoff_Weight_Bin2 THEN
                Step := 25;
            END_IF
            
        25: (* Discharge Bin 2 - OFF & Wait Transition Delay *)
            Discharge_Bin2 := FALSE;
            Transition_Timer(IN := TRUE, PT := Step_Delay_Time);
            
            IF Transition_Timer.Q AND (NOT Discharge_Bin2_Feedback OR NOT Discharge_Bin2) THEN
                Transition_Timer(IN := FALSE);
                Step := 30;
            END_IF
            
        30: (* Discharge Bin 1 - ON *)
            Discharge_Bin1 := TRUE;
            Discharge_Bin3 := FALSE;
            Discharge_Bin2 := FALSE;
            
            (* Check if current weight has dropped below target cutoff *)
            IF Current_Weight_Bin1 <= Cutoff_Weight_Bin1 THEN
                Step := 35;
            END_IF
            
        35: (* Discharge Bin 1 - OFF & Wait Transition Delay *)
            Discharge_Bin1 := FALSE;
            Transition_Timer(IN := TRUE, PT := Step_Delay_Time);
            
            IF Transition_Timer.Q AND (NOT Discharge_Bin1_Feedback OR NOT Discharge_Bin1) THEN
                Transition_Timer(IN := FALSE);
                Step := 40;
            END_IF
            
        40: (* Sequence Complete *)
            Sequence_Complete := TRUE;
            IF NOT Start_Button THEN
                Step := 0;
            END_IF
    END_CASE;

ELSE
    (* ================= MANUAL MODE ================= *)
    Step := 0;
    Sequence_Complete := FALSE;
    Transition_Timer(IN := FALSE);
    
    (* Separate manual buttons with basic interlinking *)
    IF Manual_Bin3 THEN
        Discharge_Bin3 := TRUE;
        Discharge_Bin2 := FALSE;
        Discharge_Bin1 := FALSE;
    ELSIF Manual_Bin2 THEN
        Discharge_Bin3 := FALSE;
        Discharge_Bin2 := TRUE;
        Discharge_Bin1 := FALSE;
    ELSIF Manual_Bin1 THEN
        Discharge_Bin3 := FALSE;
        Discharge_Bin2 := FALSE;
        Discharge_Bin1 := TRUE;
    ELSE
        Discharge_Bin3 := FALSE;
        Discharge_Bin2 := FALSE;
        Discharge_Bin1 := FALSE;
    END_IF;
END_IF;

END_PROGRAM

// PLC_AC500_V3/Application/old_version/batching3
PROGRAM batching3
VAR
    Step : INT := 0;          // Current active step (0: Idle, 1..6: Bins, 7: Delay, 8: Reset & Complete)
    
    (* Mode Control & Commands *)
    Start_Button : BOOL;      // Toggles process start
    E_Stop_Active : BOOL;     // Emergency Stop active signal
    
    (* Cumulative Weighing Variables *)
    load_cell_value : REAL;   // Current weight read from the single load cell
    bin_last_weight : REAL;   // Cumulative baseline weight on the load cell before starting current bin
    actual_bin : REAL;        // Current weight added from active bin
    target_act_bin : REAL;    // Target weight to add from the active bin
    bin_set_value : REAL;     // Setpoint weight for current active step
    
    (* Outputs *)
    Discharge_Bin : ARRAY[1..6] OF BOOL;
    Discharge_Bin_Feedback : ARRAY[1..6] OF BOOL;
    Actual_Weights : ARRAY[1..6] OF REAL; // Actual weight poured per silo
    Sequence_Complete : BOOL;
    
    (* RECIPE DATA STRUCTURES *)
    (* Set Weights array for 20 materials *)
    Recipe_Weights : ARRAY[1..20] OF REAL := [
        50.0,   // Material index 1 target (50.0 kg)
        15.0,   // Material index 2 target (15.0 kg)
        28.0,   // Material index 3 target (28.0 kg)
        31.0,   // Material index 4 target (31.0 kg)
        150.0,  // Material index 5 target (150.0 kg)
        10.0,   // Material index 6 target (10.0 kg)
        0.0, 0.0, 0.0, 0.0, 0.0, 0.0, 0.0, 0.0, 0.0, 0.0, 0.0, 0.0, 0.0, 0.0
    ];
    
    (* Bin Mapping for 6 Bins *)
    (* Contains 1-based Material ID index from Recipe_Weights *)
    (* If 0, the bin is skipped *)
    Bin_Material_Index : ARRAY[1..6] OF INT := [
        1,   // Bin 1 maps to Material 1 (50.0 kg)
        2,   // Bin 2 maps to Material 2 (15.0 kg)
        0,   // Bin 3 is 0 (SKIPPED)
        4,   // Bin 4 maps to Material 4 (31.0 kg)
        5,   // Bin 5 maps to Material 5 (150.0 kg)
        6    // Bin 6 maps to Material 6 (10.0 kg)
    ];
    
    Mat_Idx : INT;            // Active Material Index for lookup
    i : INT;                  // Loop index
    
    (* TIMERS FOR TRANSITIONS & DELAYS *)
    Transition_Timer : TON;
    Completion_Timer : TON;
    Step_Delay_Time : TIME := T#2S;     // Delay between closing one valve and opening the next
    Post_Complete_Delay : TIME := T#2S; // Delay after last bin closes before resetting bin_last_weight
    
    (* SELF-CONTAINED SIMULATION VARIABLES *)
    Simulation_Mode : BOOL := TRUE;
    Sim_Rate : REAL := 10.0;            // Simulated pouring speed (10.0 kg/s)
    Sim_Timer : TON;
    Start_Sim_Weight : REAL;
    Discharge_Active : BOOL;
END_VAR

(* Single Load Cell Cumulative Weighing Sequence (6 Bins with Material Mapping, Skipping, and Self-Contained Simulation) *)

(* 1. SELF-CONTAINED SIMULATION WEIGHT MANAGEMENT *)
IF Simulation_Mode THEN
    (* Reset simulation to baseline (e.g. 2.0 kg) *)
    IF Step = 0 AND NOT Start_Button AND NOT Sequence_Complete THEN
        load_cell_value := 2.0;
        bin_last_weight := 2.0;
        Start_Sim_Weight := 2.0;
        Sim_Timer(IN := FALSE);
    END_IF;
    
    (* Check if any valve is actively discharging *)
    Discharge_Active := FALSE;
    IF Step >= 1 AND Step <= 6 THEN
        Discharge_Active := Discharge_Bin[Step];
    END_IF;
    
    (* Simulate weight gain on the load cell *)
    IF Discharge_Active THEN
        Sim_Timer(IN := TRUE, PT := T#1000S);
        load_cell_value := Start_Sim_Weight + (TIME_TO_REAL(Sim_Timer.ET) / 1000.0) * Sim_Rate;
    ELSE
        Sim_Timer(IN := FALSE);
        Start_Sim_Weight := load_cell_value;
    END_IF;
END_IF;


(* 2. EMERGENCY STOP LOGIC *)
IF E_Stop_Active THEN
    FOR i := 1 TO 6 DO
        Discharge_Bin[i] := FALSE;
        Actual_Weights[i] := 0.0;
    END_FOR;
    Sequence_Complete := FALSE;
    Step := 0;
    Transition_Timer(IN := FALSE);
    Completion_Timer(IN := FALSE);
    RETURN;
END_IF;


(* 3. RECIPE START INITIALIZATION *)
IF Step = 0 AND Start_Button THEN
    Step := 1;
    bin_last_weight := load_cell_value;
    Sequence_Complete := FALSE;
    (* Clear actual weights on start *)
    FOR i := 1 TO 6 DO
        Actual_Weights[i] := 0.0;
    END_FOR;
END_IF;


(* 4. SEQUENCE CONTROL STATE MACHINE *)
CASE Step OF
    1..6: (* Discharging Silos 1 to 6 *)
        Mat_Idx := Bin_Material_Index[Step];
        
        IF Mat_Idx = 0 THEN
            (* Skip this bin instantly and step to next *)
            Step := Step + 1;
        ELSE
            (* Fetch target weight from Recipe_Weights using the mapped material index *)
            bin_set_value := Recipe_Weights[Mat_Idx];
            target_act_bin := bin_set_value;
            
            (* Calculate weight added by current active bin (increasing weight logic) *)
            actual_bin := load_cell_value - bin_last_weight;
            
            (* Update the actual weight in the array for the active bin *)
            Actual_Weights[Step] := actual_bin;
            
            (* Open discharge output valve *)
            Discharge_Bin[Step] := TRUE;
            
            (* Check if target weight has been achieved *)
            IF actual_bin >= target_act_bin THEN
                Discharge_Bin[Step] := FALSE;
                
                (* Set new baseline for the next step *)
                bin_last_weight := load_cell_value;
                
                (* Go to transition delay *)
                Step := 10 + Step; // Offset to separate transition states
            END_IF;
        END_IF;

    11..15: (* Transition Delays (Between Bins) *)
        Transition_Timer(IN := TRUE, PT := Step_Delay_Time);
        IF Transition_Timer.Q AND (NOT Discharge_Bin[Step - 10] OR NOT Discharge_Bin_Feedback[Step - 10]) THEN
            Transition_Timer(IN := FALSE);
            Step := (Step - 10) + 1; // Advance to next bin
        END_IF;
        
    16: (* Transition Delay After Last Bin (Bin 6) Closes *)
        Transition_Timer(IN := TRUE, PT := Step_Delay_Time);
        IF Transition_Timer.Q AND (NOT Discharge_Bin[6] OR NOT Discharge_Bin_Feedback[6]) THEN
            Transition_Timer(IN := FALSE);
            Step := 7; // Go to post-discharge wait step
        END_IF;

    7: (* Wait 2 Seconds After Closing the Last Bin *)
        Completion_Timer(IN := TRUE, PT := Post_Complete_Delay);
        IF Completion_Timer.Q THEN
            Completion_Timer(IN := FALSE);
            Step := 8; // Proceed to reset last weight
        END_IF;
        
    8: (* Reset bin_last_weight to 0 & Complete *)
        bin_last_weight := 0.0;
        Sequence_Complete := TRUE;
        
        IF NOT Start_Button THEN
            Step := 0;
            Sequence_Complete := FALSE;
            (* Reset all actual weights at completion once start is released *)
            FOR i := 1 TO 6 DO
                Actual_Weights[i] := 0.0;
            END_FOR;
        END_IF;
END_CASE;

END_PROGRAM

// PLC_AC500_V3/Application/old_version/batching4
PROGRAM batching4
VAR
    Step : INT := 0;          // Current active step (0: Idle, 1..6: Bins, 7: Delay, 8: Reset & Complete)
    
    (* Mode Control & Commands *)
    Start_Button : BOOL;      // Toggles process start
    E_Stop_Active : BOOL;     // Emergency Stop active signal
    
    (* Cumulative Weighing Variables *)
    load_cell_value : REAL;   // Current weight read from the single load cell
    bin_last_weight : REAL;   // Cumulative baseline weight on the load cell before starting current bin
    actual_bin : REAL;        // Current weight added from active bin
    target_act_bin : REAL;    // Target weight to add from the active bin
    bin_set_value : REAL;     // Setpoint weight for current active step
    
    (* Outputs *)
    Discharge_Bin : ARRAY[1..6] OF BOOL;
    Discharge_Bin_Feedback : ARRAY[1..6] OF BOOL;
    Actual_Weights : ARRAY[1..6] OF REAL; // Actual weight poured per silo
    Sequence_Complete : BOOL;
    
    (* RECIPE DATA STRUCTURES *)
    (* Set Weights array for 20 materials *)
    Recipe_Weights : ARRAY[1..20] OF REAL := [
        50.0,   // Material index 1 target (50.0 kg)
        15.0,   // Material index 2 target (15.0 kg)
        28.0,   // Material index 3 target (28.0 kg)
        31.0,   // Material index 4 target (31.0 kg)
        150.0,  // Material index 5 target (150.0 kg)
        10.0,   // Material index 6 target (10.0 kg)
        0.0, 0.0, 0.0, 0.0, 0.0, 0.0, 0.0, 0.0, 0.0, 0.0, 0.0, 0.0, 0.0, 0.0
    ];
    
    (* Bin Mapping for 6 Bins *)
    (* Contains 1-based Material ID index from Recipe_Weights *)
    (* If 0, the bin is skipped *)
    Bin_Material_Index : ARRAY[1..6] OF INT := [
        1,   // Bin 1 maps to Material 1 (50.0 kg)
        2,   // Bin 2 maps to Material 2 (15.0 kg)
        0,   // Bin 3 is 0 (SKIPPED)
        4,   // Bin 4 maps to Material 4 (31.0 kg)
        5,   // Bin 5 maps to Material 5 (150.0 kg)
        6    // Bin 6 maps to Material 6 (10.0 kg)
    ];
    
    Mat_Idx : INT;            // Active Material Index for lookup
    i : INT;                  // Loop index
    
    (* TIMERS FOR TRANSITIONS & DELAYS *)
    Transition_Timer : TON;
    Completion_Timer : TON;
    Step_Delay_Time : TIME := T#2S;     // Delay between closing one valve and opening the next
    Post_Complete_Delay : TIME := T#2S; // Delay after last bin closes before resetting bin_last_weight
    
    (* SELF-CONTAINED SIMULATION VARIABLES *)
    Simulation_Mode : BOOL := TRUE;
    Sim_Rate : REAL := 10.0;            // Simulated pouring speed (10.0 kg/s)
    Sim_Timer : TON;
    Start_Sim_Weight : REAL;
    Discharge_Active : BOOL;
END_VAR

(* Single Load Cell Cumulative Weighing Sequence (6 Bins with Material Mapping, Skipping, and Self-Contained Simulation) *)

(* 1. SELF-CONTAINED SIMULATION WEIGHT MANAGEMENT *)
IF Simulation_Mode THEN
    (* Reset simulation to baseline (e.g. 2.0 kg) *)
    IF Step = 0 AND NOT Start_Button AND NOT Sequence_Complete THEN
        load_cell_value := 0.0;
        bin_last_weight := 0.0;
        Start_Sim_Weight := 0.0;
        Sim_Timer(IN := FALSE);
    END_IF;
    
    (* Check if any valve is actively discharging *)
    Discharge_Active := FALSE;
    IF Step >= 1 AND Step <= 6 THEN
        Discharge_Active := Discharge_Bin[Step];
    END_IF;
    
    (* Simulate weight gain on the load cell *)
    IF Discharge_Active THEN
        Sim_Timer(IN := TRUE, PT := T#1000S);
        load_cell_value := Start_Sim_Weight + (TIME_TO_REAL(Sim_Timer.ET) / 1000.0) * Sim_Rate;
    ELSE
        Sim_Timer(IN := FALSE);
        Start_Sim_Weight := load_cell_value;
    END_IF;
END_IF;


(* 2. EMERGENCY STOP LOGIC *)
IF E_Stop_Active THEN
    FOR i := 1 TO 6 DO
        Discharge_Bin[i] := FALSE;
        Actual_Weights[i] := 0.0;
    END_FOR;
    Sequence_Complete := FALSE;
    Step := 0;
    Transition_Timer(IN := FALSE);
    Completion_Timer(IN := FALSE);
    RETURN;
END_IF;


(* 3. RECIPE START INITIALIZATION *)
IF Step = 0 AND Start_Button THEN
    Step := 1;
    bin_last_weight := load_cell_value;
    Sequence_Complete := FALSE;
    (* Clear actual weights on start *)
    FOR i := 1 TO 6 DO
        Actual_Weights[i] := 0.0;
    END_FOR;
END_IF;


(* 4. SEQUENCE CONTROL STATE MACHINE *)
CASE Step OF
    1..6: (* Discharging Silos 1 to 6 *)
        Mat_Idx := Bin_Material_Index[Step];
        
        IF Mat_Idx = 0 THEN
            (* Skip this bin instantly and step to next *)
            Step := Step + 1;
        ELSE
            (* Fetch target weight from Recipe_Weights using the mapped material index *)
            bin_set_value := Recipe_Weights[Mat_Idx];
            target_act_bin := bin_set_value;
            
            (* Calculate weight added by current active bin (increasing weight logic) *)
            actual_bin := load_cell_value - bin_last_weight;
            
            (* Update the actual weight in the array for the active bin *)
            Actual_Weights[Step] := actual_bin;
            
            (* Open discharge output valve *)
            Discharge_Bin[Step] := TRUE;
            
            (* Check if target weight has been achieved *)
            IF actual_bin >= target_act_bin THEN
                Discharge_Bin[Step] := FALSE;
                
                (* Set new baseline for the next step *)
                bin_last_weight := load_cell_value;
                
                (* Go to transition delay *)
                Step := 10 + Step; // Offset to separate transition states
            END_IF;
        END_IF;

    11..15: (* Transition Delays (Between Bins) *)
        Transition_Timer(IN := TRUE, PT := Step_Delay_Time);
        IF Transition_Timer.Q AND (NOT Discharge_Bin[Step - 10] OR NOT Discharge_Bin_Feedback[Step - 10]) THEN
            Transition_Timer(IN := FALSE);
            Step := (Step - 10) + 1; // Advance to next bin
        END_IF;
        
    16: (* Transition Delay After Last Bin (Bin 6) Closes *)
        Transition_Timer(IN := TRUE, PT := Step_Delay_Time);
        IF Transition_Timer.Q AND (NOT Discharge_Bin[6] OR NOT Discharge_Bin_Feedback[6]) THEN
            Transition_Timer(IN := FALSE);
            Step := 7; // Go to post-discharge wait step
        END_IF;

    7: (* Wait 2 Seconds After Closing the Last Bin *)
        Completion_Timer(IN := TRUE, PT := Post_Complete_Delay);
        IF Completion_Timer.Q THEN
            Completion_Timer(IN := FALSE);
            Step := 8; // Proceed to reset last weight
        END_IF;
        
    8: (* Reset bin_last_weight & Complete *)
    bin_last_weight := 0.0;
    Sequence_Complete := TRUE;

    (* Reset all actual weights *)
    FOR i := 1 TO 6 DO
        Actual_Weights[i] := 0.0;
    END_FOR;

    IF NOT Start_Button THEN
        Step := 0;
        Sequence_Complete := FALSE;
    END_IF;
END_CASE;

END_PROGRAM

// PLC_AC500_V3/Application/old_version/batching5
PROGRAM batching5
VAR
    Step : INT := 0;          // Current active step (0: Idle, 1..6: Bins, 7: Delay, 8: Reset & Complete)
    
    (* Mode Control & Commands *)
    Start_Button : BOOL;      // Toggles process start
    E_Stop_Active : BOOL;     // Emergency Stop active signal
    
    (* Cumulative Weighing Variables *)
    load_cell_value : REAL;   // Current weight read from the single load cell
    bin_last_weight : REAL;   // Cumulative baseline weight on the load cell before starting current bin
    actual_bin : REAL;        // Current weight added from active bin
    target_act_bin : REAL;    // Target weight to add from the active bin
    bin_set_value : REAL;     // Setpoint weight for current active step
    slow_cutoff_weight : REAL; // Cutoff threshold weight to switch from FAST to SLOW feed
    
    (* Dynamic Display Text *)
    Status_Message : STRING := 'System Idle';
    
    (* Outputs *)
    Discharge_Bin_Coarse : ARRAY[1..6] OF BOOL; // Coarse feed valve outputs
    Discharge_Bin_Fine : ARRAY[1..6] OF BOOL;   // Fine feed valve outputs
    Discharge_Bin_Feedback : ARRAY[1..6] OF BOOL;
    Actual_Weights : ARRAY[1..6] OF REAL; // Actual weight poured per silo
    Sequence_Complete : BOOL;
    
    (* RECIPE DATA STRUCTURES *)
    (* Set Weights array for 20 materials *)
    Recipe_Weights : ARRAY[1..20] OF REAL := [
        50.0,   // Material index 1 target (50.0 kg)
        15.0,   // Material index 2 target (15.0 kg)
        28.0,   // Material index 3 target (28.0 kg)
        31.0,   // Material index 4 target (31.0 kg)
        150.0,  // Material index 5 target (150.0 kg)
        10.0,   // Material index 6 target (10.0 kg)
        0.0, 0.0, 0.0, 0.0, 0.0, 0.0, 0.0, 0.0, 0.0, 0.0, 0.0, 0.0, 0.0, 0.0
    ];
    
    (* Set Slow Feed Transition Percentages for 20 materials *)
    (* E.g., 20.0 = Slow down when 20% of target weight is remaining *)
    Recipe_Slow_Pcts : ARRAY[1..20] OF REAL := [
        20.0,   // Silo 1: Slow down at 80% (40.0 kg)
        20.0,   // Silo 2: Slow down at 80% (12.0 kg)
        20.0,   // Silo 3: Slow down at 80%
        20.0,   // Silo 4: Slow down at 80%
        20.0,   // Silo 5: Slow down at 80%
        20.0,   // Silo 6: Slow down at 80% (8.0 kg)
        0.0, 0.0, 0.0, 0.0, 0.0, 0.0, 0.0, 0.0, 0.0, 0.0, 0.0, 0.0, 0.0, 0.0
    ];
    
    (* Bin Mapping for 6 Bins *)
    (* Contains 1-based Material ID index from Recipe_Weights *)
    (* If 0, the bin is skipped *)
    Bin_Material_Index : ARRAY[1..6] OF INT := [
        1,   // Bin 1 maps to Material 1 (50.0 kg)
        2,   // Bin 2 maps to Material 2 (15.0 kg)
        0,   // Bin 3 is 0 (SKIPPED)
        4,   // Bin 4 maps to Material 4 (31.0 kg)
        5,   // Bin 5 maps to Material 5 (150.0 kg)
        6    // Bin 6 maps to Material 6 (10.0 kg)
    ];
    
    Mat_Idx : INT;            // Active Material Index for lookup
    i : INT;                  // Loop index
    
    (* TIMERS FOR TRANSITIONS & DELAYS *)
    Transition_Timer : TON;
    Completion_Timer : TON;
    Step_Delay_Time : TIME := T#2S;     // Delay between closing one valve and opening the next
    Post_Complete_Delay : TIME := T#2S; // Delay after last bin closes before resetting bin_last_weight
    
    (* SELF-CONTAINED SIMULATION VARIABLES *)
    Simulation_Mode : BOOL := TRUE;
    Sim_Rate : REAL := 10.0;            // Simulated pouring speed (10.0 kg/s during fast feed)
    Sim_Timer : TON;
    Start_Sim_Weight : REAL;
    Discharge_Active : BOOL;
END_VAR

(* Single Load Cell Cumulative Weighing Sequence (6 Bins with Mutually Exclusive Speed Transition and Tolerance Message) *)

(* 1. SELF-CONTAINED SIMULATION WEIGHT MANAGEMENT *)
IF Simulation_Mode THEN
    (* Reset simulation to baseline (e.g. 2.0 kg) *)
    IF Step = 0 AND NOT Start_Button AND NOT Sequence_Complete THEN
        load_cell_value := 2.0;
        bin_last_weight := 2.0;
        Start_Sim_Weight := 2.0;
        Sim_Timer(IN := FALSE);
    END_IF;
    
    (* Check if any valve is actively discharging (either Coarse or Fine) *)
    Discharge_Active := FALSE;
    IF Step >= 1 AND Step <= 6 THEN
        Discharge_Active := Discharge_Bin_Coarse[Step] OR Discharge_Bin_Fine[Step];
    END_IF;
    
    (* Simulate weight gain on the load cell *)
    IF Discharge_Active THEN
        Sim_Timer(IN := TRUE, PT := T#1000S);
        load_cell_value := Start_Sim_Weight + (TIME_TO_REAL(Sim_Timer.ET) / 1000.0) * Sim_Rate;
    ELSE
        Sim_Timer(IN := FALSE);
        Start_Sim_Weight := load_cell_value;
    END_IF;
END_IF;


(* 2. EMERGENCY STOP LOGIC *)
IF E_Stop_Active THEN
    FOR i := 1 TO 6 DO
        Discharge_Bin_Coarse[i] := FALSE;
        Discharge_Bin_Fine[i] := FALSE;
        Actual_Weights[i] := 0.0;
    END_FOR;
    Sequence_Complete := FALSE;
    Step := 0;
    Status_Message := 'E-Stop Active!';
    Transition_Timer(IN := FALSE);
    Completion_Timer(IN := FALSE);
    RETURN;
END_IF;


(* 3. RECIPE START INITIALIZATION *)
IF Step = 0 AND Start_Button THEN
    Step := 1;
    bin_last_weight := load_cell_value;
    Sequence_Complete := FALSE;
    Status_Message := 'Batch Started';
    (* Clear actual weights on start *)
    FOR i := 1 TO 6 DO
        Actual_Weights[i] := 0.0;
    END_FOR;
END_IF;


(* 4. SEQUENCE CONTROL STATE MACHINE *)
CASE Step OF
    1..6: (* Discharging Silos 1 to 6 *)
        Mat_Idx := Bin_Material_Index[Step];
        
        IF Mat_Idx = 0 THEN
            (* Skip this bin instantly and step to next *)
            Step := Step + 1;
        ELSE
            (* Fetch target weight from Recipe_Weights using the mapped material index *)
            bin_set_value := Recipe_Weights[Mat_Idx];
            target_act_bin := bin_set_value;
            
            (* Calculate slow-down cutoff weight (e.g. 20% of target left) *)
            slow_cutoff_weight := target_act_bin - (target_act_bin * (Recipe_Slow_Pcts[Mat_Idx] / 100.0));
            
            (* Calculate weight added by current active bin (increasing weight logic) *)
            actual_bin := load_cell_value - bin_last_weight;
            
            (* Update the actual weight in the array for the active bin *)
            Actual_Weights[Step] := actual_bin;
            
            (* Dual-Speed Output Control & Simulation Rate Scaling *)
            IF actual_bin < slow_cutoff_weight THEN
                Discharge_Bin_Coarse[Step] := TRUE;
                Discharge_Bin_Fine[Step] := FALSE; // Mutual Exclusivity - Coarse ONLY
                Status_Message := 'Fast feeding active';
                Sim_Rate := 10.0; // Fast simulation rate
            ELSE
                Discharge_Bin_Coarse[Step] := FALSE; // Shut off coarse motor
                Discharge_Bin_Fine[Step] := TRUE;  // Mutual Exclusivity - Fine ONLY
                Status_Message := 'Tolerance weight is going on so motor is slow';
                Sim_Rate := 2.0;  // Slow simulation rate
            END_IF;
            
            (* Check if target weight has been achieved *)
            IF actual_bin >= target_act_bin THEN
                Discharge_Bin_Coarse[Step] := FALSE;
                Discharge_Bin_Fine[Step] := FALSE;
                
                (* Set new baseline for the next step *)
                bin_last_weight := load_cell_value;
                Status_Message := 'Bin Step Completed';
                
                (* Go to transition delay *)
                Step := 10 + Step; // Offset to separate transition states
            END_IF;
        END_IF;

    11..15: (* Transition Delays (Between Bins) *)
        Transition_Timer(IN := TRUE, PT := Step_Delay_Time);
        (* Verify both coarse and fine outputs are off, and feedback conforms *)
        IF Transition_Timer.Q AND (NOT Discharge_Bin_Coarse[Step - 10] AND NOT Discharge_Bin_Fine[Step - 10]) THEN
            Transition_Timer(IN := FALSE);
            Step := (Step - 10) + 1; // Advance to next bin
        END_IF;
        
    16: (* Transition Delay After Last Bin (Bin 6) Closes *)
        Transition_Timer(IN := TRUE, PT := Step_Delay_Time);
        IF Transition_Timer.Q AND (NOT Discharge_Bin_Coarse[6] AND NOT Discharge_Bin_Fine[6]) THEN
            Transition_Timer(IN := FALSE);
            Step := 7; // Go to post-discharge wait step
        END_IF;

    7: (* Wait 2 Seconds After Closing the Last Bin *)
        Status_Message := 'Settling delay active';
        Completion_Timer(IN := TRUE, PT := Post_Complete_Delay);
        IF Completion_Timer.Q THEN
            Completion_Timer(IN := FALSE);
            Step := 8; // Proceed to reset last weight
        END_IF;
        
    8: (* Reset bin_last_weight to 0 & Complete *)
        bin_last_weight := 0.0;
        Sequence_Complete := TRUE;
        Status_Message := 'Sequence Completed';
        
        IF NOT Start_Button THEN
            Step := 0;
            Sequence_Complete := FALSE;
            Status_Message := 'System Idle';
            (* Reset all actual weights at completion once start is released *)
            FOR i := 1 TO 6 DO
                Actual_Weights[i] := 0.0;
            END_FOR;
        END_IF;
END_CASE;

END_PROGRAM

// PLC_AC500_V3/Application/old_version/Auto_Batching
FUNCTION_BLOCK Auto_Batching
VAR_INPUT
    Start_Button : BOOL;      // Signal to start the batching sequence
    E_Stop_Active : BOOL;     // Emergency Stop active signal
    load_cell_value : REAL;   // Weight value read from load cell
    Discharge_Bin_Feedback : ARRAY[1..6] OF BOOL; // Physical valve feedbacks
END_VAR
VAR_OUTPUT
    Auto_Bin : ARRAY[1..6] OF BOOL; // Motor/valve control outputs
    Actual_Weights : ARRAY[1..6] OF REAL; // Actual weight poured per silo
    Sequence_Complete : BOOL;  // Batch complete flag
END_VAR
VAR
    Step : INT := 0;          // State machine index (0: Idle, 1..6: Bins, 7: Delay, 8: Reset)
    bin_last_weight : REAL;   // Baseline weight on the load cell before starting current bin
    actual_bin : REAL;        // Current weight added from active bin
    target_act_bin : REAL;    // Target weight to add from the active bin
    bin_set_value : REAL;     // Setpoint weight for current active step
    
    (* Bin Mapping for 6 Auto Bins *)
    (* Maps physical Silo 1..6 to Material Index 1..20 *)
    Bin_Material_Index : ARRAY[1..6] OF INT := [
        1,   // Bin 1 maps to Material 1 (50.0 kg)
        2,   // Bin 2 maps to Material 2 (15.0 kg)
        0,   // Bin 3 is 0 (SKIPPED)
        4,   // Bin 4 maps to Material 4 (31.0 kg)
        5,   // Bin 5 maps to Material 5 (150.0 kg)
        6    // Bin 6 maps to Material 6 (10.0 kg)
    ];
    
    Mat_Idx : INT;
    i : INT;                  // General loop index
    
    (* TIMERS FOR TRANSITIONS & DELAYS *)
    Transition_Timer : TON;
    Completion_Timer : TON;
    Step_Delay_Time : TIME := T#2S;
    Post_Complete_Delay : TIME := T#2S;
    
    (* SELF-CONTAINED SIMULATION VARIABLES *)
    Simulation_Mode : BOOL := TRUE;
    Sim_Rate : REAL := 10.0;            // Simulated pouring speed (10.0 kg/s)
    Sim_Timer : TON;
    Start_Sim_Weight : REAL;
    Discharge_Active : BOOL;
END_VAR

(* Cumulative Gain-in-Weight Auto Batching FB *)

(* 1. SELF-CONTAINED SIMULATION WEIGHT MANAGEMENT *)
IF Simulation_Mode THEN
    (* Reset simulation to baseline (e.g. 2.0 kg) *)
    IF Step = 0 AND NOT Start_Button AND NOT Sequence_Complete THEN
        load_cell_value := 2.0;
        bin_last_weight := 2.0;
        Start_Sim_Weight := 2.0;
        Sim_Timer(IN := FALSE);
    END_IF;
    
    (* Check if any valve is actively discharging *)
    Discharge_Active := FALSE;
    IF Step >= 1 AND Step <= 6 THEN
        Discharge_Active := Auto_Bin[Step];
    END_IF;
    
    (* Simulate weight gain on the load cell *)
    IF Discharge_Active THEN
        Sim_Timer(IN := TRUE, PT := T#1000S);
        load_cell_value := Start_Sim_Weight + (TIME_TO_REAL(Sim_Timer.ET) / 1000.0) * Sim_Rate;
    ELSE
        Sim_Timer(IN := FALSE);
        Start_Sim_Weight := load_cell_value;
    END_IF;
END_IF;


(* 2. EMERGENCY STOP LOGIC *)
IF E_Stop_Active THEN
    FOR i := 1 TO 6 DO
        Auto_Bin[i] := FALSE;
        Actual_Weights[i] := 0.0;
    END_FOR;
    Sequence_Complete := FALSE;
    Step := 0;
    Transition_Timer(IN := FALSE);
    Completion_Timer(IN := FALSE);
    RETURN;
END_IF;


(* 3. RECIPE SEQUENCE START *)
IF Step = 0 AND Start_Button THEN
    Step := 1;
    bin_last_weight := load_cell_value;
    Sequence_Complete := FALSE;
    (* Clear actual weights on start *)
    FOR i := 1 TO 6 DO
        Actual_Weights[i] := 0.0;
    END_FOR;
END_IF;


(* 4. SEQUENCE CONTROL STATE MACHINE *)
CASE Step OF
    1..6: (* Discharging Silos 1 to 6 *)
        Mat_Idx := Bin_Material_Index[Step];
        
        IF Mat_Idx = 0 THEN
            (* Skip this bin instantly *)
            Step := Step + 1;
        ELSE
            (* Fetch target weight from global Recipe_Weights array *)
            bin_set_value := GVL.Recipe_Weights[Mat_Idx];
            target_act_bin := bin_set_value;
            
            (* Calculate weight added by current active bin *)
            actual_bin := load_cell_value - bin_last_weight;
            
            (* Update the actual weight in the array for the active bin *)
            Actual_Weights[Step] := actual_bin;
            
            (* Open discharge output valve *)
            Auto_Bin[Step] := TRUE;
            
            (* Check if target weight has been achieved *)
            IF actual_bin >= target_act_bin THEN
                Auto_Bin[Step] := FALSE;
                
                (* Set new baseline for the next step *)
                bin_last_weight := load_cell_value;
                
                (* Go to transition delay *)
                Step := 10 + Step; // Offset to separate transition states
            END_IF;
        END_IF;

    11..15: (* Transition Delays (Between Bins) *)
        Transition_Timer(IN := TRUE, PT := Step_Delay_Time);
        IF Transition_Timer.Q AND (NOT Auto_Bin[Step - 10] OR NOT Discharge_Bin_Feedback[Step - 10]) THEN
            Transition_Timer(IN := FALSE);
            Step := (Step - 10) + 1; // Advance to next bin
        END_IF;
        
    16: (* Transition Delay After Last Bin (Bin 6) Closes *)
        Transition_Timer(IN := TRUE, PT := Step_Delay_Time);
        IF Transition_Timer.Q AND (NOT Auto_Bin[6] OR NOT Discharge_Bin_Feedback[6]) THEN
            Transition_Timer(IN := FALSE);
            Step := 7; // Go to post-discharge wait step
        END_IF;

    7: (* Wait 2 Seconds After Closing the Last Bin *)
        Completion_Timer(IN := TRUE, PT := Post_Complete_Delay);
        IF Completion_Timer.Q THEN
            Completion_Timer(IN := FALSE);
            Step := 8; // Proceed to reset last weight
        END_IF;
        
    8: (* Reset bin_last_weight to 0 & Complete *)
        bin_last_weight := 0.0;
        Sequence_Complete := TRUE;
        
        IF NOT Start_Button THEN
            Step := 0;
            Sequence_Complete := FALSE;
            (* Reset all actual weights at completion once start is released *)
            FOR i := 1 TO 6 DO
                Actual_Weights[i] := 0.0;
            END_FOR;
        END_IF;
END_CASE;

END_FUNCTION_BLOCK

// PLC_AC500_V3/Application/old_version/Manual_Batching
FUNCTION_BLOCK Manual_Batching
VAR_INPUT
    Start_Button : BOOL;      // Signal to start the batching sequence
    E_Stop_Active : BOOL;     // Emergency Stop active signal
    load_cell_value : REAL;   // Weight value read from load cell
END_VAR
VAR_OUTPUT
    Manual_Bin : ARRAY[1..10] OF BOOL; // Prompts/indicators for Bins 7..16
    Actual_Weights : ARRAY[1..10] OF REAL; // Actual weight poured per silo
    Sequence_Complete : BOOL;  // Batch complete flag
END_VAR
VAR
    Step : INT := 0;          // State machine index (0: Idle, 1..10: Bins, 11..20: Delays, 30: Settling, 40: Complete)
    bin_last_weight : REAL;   // Baseline weight on the load cell before starting current bin
    actual_bin : REAL;        // Current weight added from active bin
    target_act_bin : REAL;    // Target weight to add from the active bin
    bin_set_value : REAL;     // Setpoint weight for current active step
    
    (* Bin Mapping for 10 Manual Bins *)
    (* Maps physical manual Silo 7..16 to Material Index 1..20 *)
    Bin_Manual_Index : ARRAY[1..10] OF INT := [
        7,    // Silo 7 maps to Material 7 (12.0 kg)
        8,    // Silo 8 maps to Material 8 (8.0 kg)
        0,    // Silo 9 is 0 (SKIPPED)
        10,   // Silo 10 maps to Material 10 (5.0 kg)
        11,   // Silo 11 maps to Material 11 (18.0 kg)
        12,   // Silo 12 maps to Material 12 (22.0 kg)
        13,   // Silo 13 maps to Material 13 (30.0 kg)
        14,   // Silo 14 maps to Material 14 (14.0 kg)
        15,   // Silo 15 maps to Material 15 (9.0 kg)
        16    // Silo 16 maps to Material 16 (11.0 kg)
    ];
    
    Mat_Idx : INT;
    i : INT;                  // General loop index
    
    (* TIMERS FOR TRANSITIONS & DELAYS *)
    Transition_Timer : TON;
    Completion_Timer : TON;
    Step_Delay_Time : TIME := T#2S;
    Post_Complete_Delay : TIME := T#2S;
    
    (* SELF-CONTAINED SIMULATION VARIABLES *)
    Simulation_Mode : BOOL := TRUE;
    Sim_Rate : REAL := 10.0;            // Simulated pouring speed (10.0 kg/s)
    Sim_Timer : TON;
    Start_Sim_Weight : REAL;
    Discharge_Active : BOOL;
END_VAR

(* Cumulative Gain-in-Weight Manual Batching FB (Simulates Operator Pouring) *)

(* 1. SIMULATION WEIGHT MANAGEMENT *)
IF Simulation_Mode THEN
    (* Reset simulation to baseline (e.g. 2.0 kg) *)
    IF Step = 0 AND NOT Start_Button AND NOT Sequence_Complete THEN
        load_cell_value := 2.0;
        bin_last_weight := 2.0;
        Start_Sim_Weight := 2.0;
        Sim_Timer(IN := FALSE);
    END_IF;
    
    (* Check if operator is actively pouring *)
    Discharge_Active := FALSE;
    IF Step >= 1 AND Step <= 10 THEN
        Discharge_Active := Manual_Bin[Step];
    END_IF;
    
    (* Simulate weight gain on the load cell *)
    IF Discharge_Active THEN
        Sim_Timer(IN := TRUE, PT := T#1000S);
        load_cell_value := Start_Sim_Weight + (TIME_TO_REAL(Sim_Timer.ET) / 1000.0) * Sim_Rate;
    ELSE
        Sim_Timer(IN := FALSE);
        Start_Sim_Weight := load_cell_value;
    END_IF;
END_IF;


(* 2. EMERGENCY STOP LOGIC *)
IF E_Stop_Active THEN
    FOR i := 1 TO 10 DO
        Manual_Bin[i] := FALSE;
        Actual_Weights[i] := 0.0;
    END_FOR;
    Sequence_Complete := FALSE;
    Step := 0;
    Transition_Timer(IN := FALSE);
    Completion_Timer(IN := FALSE);
    RETURN;
END_IF;


(* 3. RECIPE SEQUENCE START *)
IF Step = 0 AND Start_Button THEN
    Step := 1;
    bin_last_weight := load_cell_value;
    Sequence_Complete := FALSE;
    (* Clear actual weights on start *)
    FOR i := 1 TO 10 DO
        Actual_Weights[i] := 0.0;
    END_FOR;
END_IF;


(* 4. SEQUENCE CONTROL STATE MACHINE *)
CASE Step OF
    1..10: (* Prompts Silos 7 to 16 *)
        Mat_Idx := Bin_Manual_Index[Step];
        
        IF Mat_Idx = 0 THEN
            (* Skip this bin instantly *)
            Step := Step + 1;
        ELSE
            (* Fetch target weight from global Recipe_Weights array *)
            bin_set_value := GVL.Recipe_Weights[Mat_Idx];
            target_act_bin := bin_set_value;
            
            (* Calculate weight added by current active bin *)
            actual_bin := load_cell_value - bin_last_weight;
            
            (* Update the actual weight in the array for the active bin *)
            Actual_Weights[Step] := actual_bin;
            
            (* Prompt operator indicator active *)
            Manual_Bin[Step] := TRUE;
            
            (* Check if target weight has been achieved *)
            IF actual_bin >= target_act_bin THEN
                Manual_Bin[Step] := FALSE;
                
                (* Set new baseline for the next step *)
                bin_last_weight := load_cell_value;
                
                (* Go to transition delay *)
                Step := 10 + Step; // Offset to separate transition states
            END_IF;
        END_IF;

    11..19: (* Transition Delays (Between Bins) *)
        Transition_Timer(IN := TRUE, PT := Step_Delay_Time);
        IF Transition_Timer.Q THEN
            Transition_Timer(IN := FALSE);
            Step := (Step - 10) + 1; // Advance to next bin
        END_IF;
        
    20: (* Transition Delay After Last Bin (Bin 10) Closes *)
        Transition_Timer(IN := TRUE, PT := Step_Delay_Time);
        IF Transition_Timer.Q THEN
            Transition_Timer(IN := FALSE);
            Step := 30; // Go to post-discharge wait step (State 30)
        END_IF;

    30: (* Wait 2 Seconds After Closing the Last Bin *)
        Completion_Timer(IN := TRUE, PT := Post_Complete_Delay);
        IF Completion_Timer.Q THEN
            Completion_Timer(IN := FALSE);
            Step := 40; // Proceed to reset last weight (State 40)
        END_IF;
        
    40: (* Reset bin_last_weight to 0 & Complete *)
        bin_last_weight := 0.0;
        Sequence_Complete := TRUE;
        
        IF NOT Start_Button THEN
            Step := 0;
            Sequence_Complete := FALSE;
            (* Reset all actual weights at completion once start is released *)
            FOR i := 1 TO 10 DO
                Actual_Weights[i] := 0.0;
            END_FOR;
        END_IF;
END_CASE;

END_FUNCTION_BLOCK

// PLC_AC500_V3/Application/old_version/batching6
PROGRAM batching6
VAR
    Auto_Ctrl : Auto_Batching;
    Manual_Ctrl : Manual_Batching;
    
    (* Global Inputs & Toggles *)
    Start_Button : BOOL;
    E_Stop_Active : BOOL;
    
    (* Parallel Weight Feedbacks *)
    load_cell_auto : REAL;
    load_cell_manual : REAL;
    
    (* Process Outputs *)
    Auto_Bin : ARRAY[1..6] OF BOOL;
    Manual_Bin : ARRAY[1..10] OF BOOL;
    
    Auto_Weights : ARRAY[1..6] OF REAL;
    Manual_Weights : ARRAY[1..10] OF REAL;
    
    Auto_Complete : BOOL;
    Manual_Complete : BOOL;
    Sequence_Complete : BOOL;
END_VAR

(* Run Auto & Manual Batching pipelines concurrently in parallel *)

Auto_Ctrl(
    Start_Button := Start_Button,
    E_Stop_Active := E_Stop_Active,
    load_cell_value := load_cell_auto,
    Discharge_Bin_Feedback := ,
    Auto_Bin => Auto_Bin,
    Actual_Weights => Auto_Weights,
    Sequence_Complete => Auto_Complete
);

Manual_Ctrl(
    Start_Button := Start_Button,
    E_Stop_Active := E_Stop_Active,
    load_cell_value := load_cell_manual,
    Manual_Bin => Manual_Bin,
    Actual_Weights => Manual_Weights,
    Sequence_Complete => Manual_Complete
);

(* Global complete once both streams conclude *)
Sequence_Complete := Auto_Complete AND Manual_Complete;

END_PROGRAM

// PLC_AC500_V3/Application/old_version/Auto_Batching_V7
FUNCTION_BLOCK Auto_Batching_V7
VAR_INPUT
    Start_Button : BOOL;      // Signal to start the batching sequence
    E_Stop_Active : BOOL;     // Emergency Stop active signal
    load_cell_value : REAL;   // Weight value read from load cell
    Discharge_Bin_Feedback : ARRAY[1..6] OF BOOL; // Physical valve feedbacks
    Bin_Material_Index : ARRAY[1..6] OF INT;      // Mapped material index inputs
END_VAR
VAR_OUTPUT
    Auto_Bin : ARRAY[1..6] OF BOOL; // Motor/valve control outputs
    Actual_Weights : ARRAY[1..6] OF REAL; // Actual weight poured per silo
    Sequence_Complete : BOOL;  // Batch complete flag
    Active_Material_ID : INT;  // Currently active ingredient ID
    Active_Bin_ID : INT;       // Currently active physical Bin ID (1..6)
END_VAR
VAR
    Step : INT := 0;          // State machine index (0: Idle, 1..6: Bins, 7: Delay, 8: Reset)
    bin_last_weight : REAL;   // Baseline weight on the load cell before starting current bin
    actual_bin : REAL;        // Current weight added from active bin
    target_act_bin : REAL;    // Target weight to add from the active bin
    bin_set_value : REAL;     // Setpoint weight for current active step
    
    Mat_Idx : INT;
    i : INT;                  // General loop index
    
    (* TIMERS FOR TRANSITIONS & DELAYS *)
    Transition_Timer : TON;
    Completion_Timer : TON;
    Step_Delay_Time : TIME := T#2S;
    Post_Complete_Delay : TIME := T#2S;
    
    (* SELF-CONTAINED SIMULATION VARIABLES *)
    Simulation_Mode : BOOL := TRUE;
    Sim_Rate : REAL := 10.0;            // Simulated pouring speed (10.0 kg/s)
    Sim_Timer : TON;
    Start_Sim_Weight : REAL;
    Discharge_Active : BOOL;
END_VAR

(* Cumulative Gain-in-Weight Auto Batching FB V7 *)

(* 1. SELF-CONTAINED SIMULATION WEIGHT MANAGEMENT *)
IF Simulation_Mode THEN
    (* Reset simulation to baseline (e.g. 2.0 kg) *)
    IF Step = 0 AND NOT Start_Button AND NOT Sequence_Complete THEN
        load_cell_value := 2.0;
        bin_last_weight := 2.0;
        Start_Sim_Weight := 2.0;
        Sim_Timer(IN := FALSE);
    END_IF;
    
    (* Check if any valve is actively discharging *)
    Discharge_Active := FALSE;
    IF Step >= 1 AND Step <= 6 THEN
        Discharge_Active := Auto_Bin[Step];
    END_IF;
    
    (* Simulate weight gain on the load cell *)
    IF Discharge_Active THEN
        Sim_Timer(IN := TRUE, PT := T#1000S);
        load_cell_value := Start_Sim_Weight + (TIME_TO_REAL(Sim_Timer.ET) / 1000.0) * Sim_Rate;
    ELSE
        Sim_Timer(IN := FALSE);
        Start_Sim_Weight := load_cell_value;
    END_IF;
END_IF;


(* 2. EMERGENCY STOP LOGIC *)
IF E_Stop_Active THEN
    FOR i := 1 TO 6 DO
        Auto_Bin[i] := FALSE;
        Actual_Weights[i] := 0.0;
    END_FOR;
    Sequence_Complete := FALSE;
    Step := 0;
    Active_Material_ID := 0;
    Active_Bin_ID := 0;
    Transition_Timer(IN := FALSE);
    Completion_Timer(IN := FALSE);
    RETURN;
END_IF;


(* 3. RECIPE SEQUENCE START *)
IF Step = 0 AND Start_Button THEN
    Step := 1;
    bin_last_weight := load_cell_value;
    Sequence_Complete := FALSE;
    (* Clear actual weights on start *)
    FOR i := 1 TO 6 DO
        Actual_Weights[i] := 0.0;
    END_FOR;
END_IF;


(* 4. SEQUENCE CONTROL STATE MACHINE *)
CASE Step OF
    0:
        Active_Material_ID := 0;
        Active_Bin_ID := 0;
        
    1..6: (* Discharging Silos 1 to 6 *)
        Mat_Idx := Bin_Material_Index[Step];
        
        IF Mat_Idx = 0 THEN
            (* Skip this bin instantly *)
            Step := Step + 1;
        ELSE
            (* Fetch target weight from global Recipe_Weights array *)
            bin_set_value := GVL.Recipe_Weights[Mat_Idx];
            target_act_bin := bin_set_value;
            
            (* Calculate weight added by current active bin *)
            actual_bin := load_cell_value - bin_last_weight;
            
            (* Update the actual weight in the array for the active bin *)
            Actual_Weights[Step] := actual_bin;
            
            (* Open discharge output valve *)
            Auto_Bin[Step] := TRUE;
            
            (* Output currently active IDs *)
            Active_Material_ID := Mat_Idx;
            Active_Bin_ID := Step;
            
            (* Check if target weight has been achieved *)
            IF actual_bin >= target_act_bin THEN
                Auto_Bin[Step] := FALSE;
                
                (* Set new baseline for the next step *)
                bin_last_weight := load_cell_value;
                
                (* Go to transition delay *)
                Step := 10 + Step; // Offset to separate transition states
            END_IF;
        END_IF;

    11..15: (* Transition Delays (Between Bins) *)
        Active_Material_ID := 0;
        Active_Bin_ID := 0;
        Transition_Timer(IN := TRUE, PT := Step_Delay_Time);
        IF Transition_Timer.Q AND (NOT Auto_Bin[Step - 10] OR NOT Discharge_Bin_Feedback[Step - 10]) THEN
            Transition_Timer(IN := FALSE);
            Step := (Step - 10) + 1; // Advance to next bin
        END_IF;
        
    16: (* Transition Delay After Last Bin (Bin 6) Closes *)
        Active_Material_ID := 0;
        Active_Bin_ID := 0;
        Transition_Timer(IN := TRUE, PT := Step_Delay_Time);
        IF Transition_Timer.Q AND (NOT Auto_Bin[6] OR NOT Discharge_Bin_Feedback[6]) THEN
            Transition_Timer(IN := FALSE);
            Step := 7; // Go to post-discharge wait step
        END_IF;

    7: (* Wait 2 Seconds After Closing the Last Bin *)
        Active_Material_ID := 0;
        Active_Bin_ID := 0;
        Completion_Timer(IN := TRUE, PT := Post_Complete_Delay);
        IF Completion_Timer.Q THEN
            Completion_Timer(IN := FALSE);
            Step := 8; // Proceed to reset last weight
        END_IF;
        
    8: (* Reset bin_last_weight to 0 & Complete *)
        Active_Material_ID := 0;
        Active_Bin_ID := 0;
        bin_last_weight := 0.0;
        Sequence_Complete := TRUE;
        
        IF NOT Start_Button THEN
            Step := 0;
            Sequence_Complete := FALSE;
            (* Reset all actual weights at completion once start is released *)
            FOR i := 1 TO 6 DO
                Actual_Weights[i] := 0.0;
            END_FOR;
        END_IF;
END_CASE;

END_FUNCTION_BLOCK

// PLC_AC500_V3/Application/old_version/Manual_Batching_V7
FUNCTION_BLOCK Manual_Batching_V7
VAR_INPUT
    Start_Button : BOOL;      // Signal to start the batching sequence
    E_Stop_Active : BOOL;     // Emergency Stop active signal
    load_cell_value : REAL;   // Weight value read from load cell
    Bin_Manual_Index : ARRAY[1..10] OF INT; // Mapped material index inputs
END_VAR
VAR_OUTPUT
    Manual_Bin : ARRAY[1..10] OF BOOL; // Prompts/indicators for Bins 7..16
    Actual_Weights : ARRAY[1..10] OF REAL; // Actual weight poured per silo
    Sequence_Complete : BOOL;  // Batch complete flag
    Active_Material_ID : INT;  // Currently active ingredient ID
    Active_Bin_ID : INT;       // Currently active physical Bin ID (7..16)
END_VAR
VAR
    Step : INT := 0;          // State machine index (0: Idle, 1..10: Bins, 11..20: Delays, 30: Settling, 40: Complete)
    bin_last_weight : REAL;   // Baseline weight on the load cell before starting current bin
    actual_bin : REAL;        // Current weight added from active bin
    target_act_bin : REAL;    // Target weight to add from the active bin
    bin_set_value : REAL;     // Setpoint weight for current active step
    
    Mat_Idx : INT;
    i : INT;                  // General loop index
    
    (* TIMERS FOR TRANSITIONS & DELAYS *)
    Transition_Timer : TON;
    Completion_Timer : TON;
    Step_Delay_Time : TIME := T#2S;
    Post_Complete_Delay : TIME := T#2S;
    
    (* SELF-CONTAINED SIMULATION VARIABLES *)
    Simulation_Mode : BOOL := TRUE;
    Sim_Rate : REAL := 10.0;            // Simulated pouring speed (10.0 kg/s)
    Sim_Timer : TON;
    Start_Sim_Weight : REAL;
    Discharge_Active : BOOL;
END_VAR

(* Cumulative Gain-in-Weight Manual Batching FB V7 *)

(* 1. SIMULATION WEIGHT MANAGEMENT *)
IF Simulation_Mode THEN
    (* Reset simulation to baseline (e.g. 2.0 kg) *)
    IF Step = 0 AND NOT Start_Button AND NOT Sequence_Complete THEN
        load_cell_value := 2.0;
        bin_last_weight := 2.0;
        Start_Sim_Weight := 2.0;
        Sim_Timer(IN := FALSE);
    END_IF;
    
    (* Check if operator is actively pouring *)
    Discharge_Active := FALSE;
    IF Step >= 1 AND Step <= 10 THEN
        Discharge_Active := Manual_Bin[Step];
    END_IF;
    
    (* Simulate weight gain on the load cell *)
    IF Discharge_Active THEN
        Sim_Timer(IN := TRUE, PT := T#1000S);
        load_cell_value := Start_Sim_Weight + (TIME_TO_REAL(Sim_Timer.ET) / 1000.0) * Sim_Rate;
    ELSE
        Sim_Timer(IN := FALSE);
        Start_Sim_Weight := load_cell_value;
    END_IF;
END_IF;


(* 2. EMERGENCY STOP LOGIC *)
IF E_Stop_Active THEN
    FOR i := 1 TO 10 DO
        Manual_Bin[i] := FALSE;
        Actual_Weights[i] := 0.0;
    END_FOR;
    Sequence_Complete := FALSE;
    Step := 0;
    Active_Material_ID := 0;
    Active_Bin_ID := 0;
    Transition_Timer(IN := FALSE);
    Completion_Timer(IN := FALSE);
    RETURN;
END_IF;


(* 3. RECIPE SEQUENCE START *)
IF Step = 0 AND Start_Button THEN
    Step := 1;
    bin_last_weight := load_cell_value;
    Sequence_Complete := FALSE;
    (* Clear actual weights on start *)
    FOR i := 1 TO 10 DO
        Actual_Weights[i] := 0.0;
    END_FOR;
END_IF;


(* 4. SEQUENCE CONTROL STATE MACHINE *)
CASE Step OF
    0:
        Active_Material_ID := 0;
        Active_Bin_ID := 0;
        
    1..10: (* Prompts Silos 7 to 16 *)
        Mat_Idx := Bin_Manual_Index[Step];
        
        IF Mat_Idx = 0 THEN
            (* Skip this bin instantly *)
            Step := Step + 1;
        ELSE
            (* Fetch target weight from global Recipe_Weights array *)
            bin_set_value := GVL.Recipe_Weights[Mat_Idx];
            target_act_bin := bin_set_value;
            
            (* Calculate weight added by current active bin *)
            actual_bin := load_cell_value - bin_last_weight;
            
            (* Update the actual weight in the array for the active bin *)
            Actual_Weights[Step] := actual_bin;
            
            (* Prompt operator indicator active *)
            Manual_Bin[Step] := TRUE;
            
            (* Output currently active IDs (Shift to physical Silo ID 7..16) *)
            Active_Material_ID := Mat_Idx;
            Active_Bin_ID := Step;
            
            (* Check if target weight has been achieved *)
            IF actual_bin >= target_act_bin THEN
                Manual_Bin[Step] := FALSE;
                
                (* Set new baseline for the next step *)
                bin_last_weight := load_cell_value;
                
                (* Go to transition delay *)
                Step := 10 + Step; // Offset to separate transition states
            END_IF;
        END_IF;

    11..19: (* Transition Delays (Between Bins) *)
        Active_Material_ID := 0;
        Active_Bin_ID := 0;
        Transition_Timer(IN := TRUE, PT := Step_Delay_Time);
        IF Transition_Timer.Q THEN
            Transition_Timer(IN := FALSE);
            Step := (Step - 10) + 1; // Advance to next bin
        END_IF;
        
    20: (* Transition Delay After Last Bin (Bin 10) Closes *)
        Active_Material_ID := 0;
        Active_Bin_ID := 0;
        Transition_Timer(IN := TRUE, PT := Step_Delay_Time);
        IF Transition_Timer.Q THEN
            Transition_Timer(IN := FALSE);
            Step := 30; // Go to post-discharge wait step (State 30)
        END_IF;

    30: (* Wait 2 Seconds After Closing the Last Bin *)
        Active_Material_ID := 0;
        Active_Bin_ID := 0;
        Completion_Timer(IN := TRUE, PT := Post_Complete_Delay);
        IF Completion_Timer.Q THEN
            Completion_Timer(IN := FALSE);
            Step := 40; // Proceed to reset last weight (State 40)
        END_IF;
        
    40: (* Reset bin_last_weight to 0 & Complete *)
        Active_Material_ID := 0;
        Active_Bin_ID := 0;
        bin_last_weight := 0.0;
        Sequence_Complete := TRUE;
        
        IF NOT Start_Button THEN
            Step := 0;
            Sequence_Complete := FALSE;
            (* Reset all actual weights at completion once start is released *)
            FOR i := 1 TO 10 DO
                Actual_Weights[i] := 0.0;
            END_FOR;
        END_IF;
END_CASE;

END_FUNCTION_BLOCK

// PLC_AC500_V3/Application/old_version/batching7
PROGRAM batching7
VAR
    Auto_Ctrl : Auto_Batching_V7;
    Manual_Ctrl : Manual_Batching_V7;
    
    (* Global Inputs & Toggles *)
    Start_Button : BOOL;
    E_Stop_Active : BOOL;
    
    (* Parallel Weight Feedbacks *)
    load_cell_auto : REAL;
    load_cell_manual : REAL;
    
    (* Process Outputs *)
    Auto_Bin : ARRAY[1..6] OF BOOL;
    Manual_Bin : ARRAY[1..10] OF BOOL;
    
    Auto_Weights : ARRAY[1..6] OF REAL;
    Manual_Weights : ARRAY[1..10] OF REAL;
    
    Auto_Complete : BOOL;
    Manual_Complete : BOOL;
    Sequence_Complete : BOOL;
    
